(* CoDeSys 2.3.9.16 project: oscat320.pro *)
(* Libraries: Standard.lib 22.11.04 10:21:12 *)

(* PLC configuration (modules and I/O channels)
K-Bus [K_Bus] node 0, in %IB0 out %QB0
Fieldbus variables [FB_VARS] node 1, in %IB0 out %QB0
*)

(* Global variable list: Constants *)
VAR_GLOBAL CONSTANT
	STRING_LENGTH : INT := 250;
	NETWORK_BUFFER_LONG_SIZE : UINT := 3999;
	NETWORK_BUFFER_SHORT_SIZE : UINT := 1459;
END_VAR




(* revisionhistory
hm 3. mar. 2007
	extended accuracy of pi2
	renamed T0 to Tk for better compatibility with other libraries
	renamed C t0 c0 for better compatibility

hm	2. may. 2007
	added RU universal gas constant

hm	1. oct. 2007
	added setup parameter STEP7

hm 31. oct. 2007
	added PN

hm	6. mar. 2008
	added setup Parameter EXTENDED_ASCII

hm	28. Mar. 2008
	added setup parameter STRING_LENGTH

hm	7. apr. 2008
	Deleted unused setup parameter Step7

hm	19. apr. 2008
	added setup parameter NETWORK_BUFFER_SIZE

hm	27. apr. 2008
	added PI05 and PI025

hm	18. may. 2008
	added charname lists
	renamed E to E1

hm	30. jun. 2008
	reduced size of string constants to 253 to avoid problems with target aixia DCUF

hm	21. sep. 2008
	added section language setup
	added section location setup

hm	20. oct. 2008
	changed to structured constants

hm	16. nov. 2008
	moved structured constants to global vars for compatibility reasons

hm	13. nov. 2009
	added network_buffer_short_size
	renamed network_buffer_long_size
	changed string length to 250
*)

(* Global variable list: Globale_Variablen *)
VAR_GLOBAL
	MATH : CONSTANTS_MATH;
	PHYS : CONSTANTS_PHYS;
	LANGUAGE : CONSTANTS_LANGUAGE;
	SETUP : CONSTANTS_SETUP;
	LOCATION : CONSTANTS_LOCATION;
END_VAR

(* Data type *)
TYPE CALENDAR :
STRUCT
	UTC : DT;						(* world time UTC *)
	LDT : DT;						(* local time *)
	LDATE : DATE;				(* local date *)
	LTOD : TOD;					(* local time of day *)
	YEAR : INT;					(* year of LDATE *)
	MONTH : INT;					(* month of LDATE *)
	DAY : INT;						(* day of LDATE *)
	WEEKDAY : INT;				(* weekday of LDATE *)
	OFFSET : INT;					(* Time Zone Offset for Local time in minutes *)
	DST_EN : BOOL;				(* daylight savings time enable *)
	DST_ON : BOOL;				(* true when daylight savings time os on *)
	NAME : STRING(5);			(* name of time zone *)
	LOCATION : INT;				(* location number pls see location setup *)
	LONGITUDE : REAL;			(* longitude of current location *)
	LATITUDE : REAL;			(* latitude of current location *)
	SUN_RISE : TOD;				(* sun_rise for current location *)
	SUN_SET : TOD;				(* sun_set for current location *)
	SUN_MIDDAY : TOD;			(* worldtime when sun stands at south position *)
	SUN_HEIGTH : REAL	;		(* suns heigth at midday, south position *)
	SUN_HOR : REAL;			(* sun angle horizontal 0 = north in degrees *)
	SUN_VER : REAL;			(* sun angle vertical above horizon in degrees *)
	NIGHT : BOOL;				(* true between sun_set and sun_rise *)
	HOLIDAY : BOOL;				(* true when holiday *)
	HOLY_NAME : STRING(30);	(* name of holiday *)
	WORK_WEEK : INT;			(* current work week *)
END_STRUCT
END_TYPE

(* revision history
hm	21. nov. 2008	rev 1.0
	original version

hm	8. feb. 2009	rev 1.1
	added sun position data

hm	10. mar. 2009	rev 1.2
	added work_week, sun_midday, sun_heigth
*)

(* Data type *)
TYPE COMPLEX :
STRUCT
	re : REAL;
	im : REAL;
END_STRUCT
END_TYPE


(* revision history
hm	18. oct. 2008
	original version

*)

(* Data type *)
TYPE CONSTANTS_LANGUAGE :
STRUCT
	(* Language Setup *)
	DEFAULT : INT := 1; (* 1=english, 2=german 3=french *)
	LMAX : INT := 3;
	WEEKDAYS : ARRAY[1..3, 1..7] OF STRING(10) :=	'Monday', 'Tuesday', 'Wednesday', 'Thursday', 'Friday', 'Saturday', 'Sunday',
													'Montag', 'Dienstag', 'Mittwoch', 'Donnerstag', 'Freitag', 'Samstag', 'Sonntag',
													'Lundi', 'Mardi', 'Mercredi', 'Jeudi', 'Vendredi', 'Samedi', 'Dimanche';
	WEEKDAYS2 : ARRAY[1..3, 1..7] OF STRING(2) :=	'Mo', 'Tu', 'We', 'Th', 'Fr', 'Sa', 'Su',
													'Mo', 'Di', 'Mi', 'Do', 'Fr', 'Sa', 'So',
													'Lu', 'Ma', 'Me', 'Je', 'Ve', 'Sa', 'Di';
	MONTHS : ARRAY[1..3, 1..12] OF STRING(10) :=	'January', 'February', 'March', 'April', 'May', 'June', 'July', 'August', 'September', 'October', 'November', 'December',
													'Januar', 'Februar', 'März', 'April', 'Mai', 'Juni', 'Juli', 'August', 'September', 'Oktober', 'November', 'Dezember',
													'Janvier', 'Février', 'mars', 'Avril', 'Mai', 'Juin', 'Juillet', 'Août', 'Septembre', 'Octobre', 'Novembre', 'Decembre';
	MONTHS3 : ARRAY[1..3, 1..12] OF STRING(3) :=	'Jan', 'Feb', 'Mar', 'Apr', 'May', 'Jun', 'Jul', 'Aug', 'Sep', 'Oct', 'Nov', 'Dec',
													'Jan', 'Feb', 'Mrz', 'Apr', 'Mai', 'Jun', 'Jul', 'Aug', 'Sep', 'Okt', 'Nov', 'Dez',
													'Jan', 'Fev', 'Mar', 'Avr', 'Mai', 'Jun', 'Jul', 'Aou', 'Sep', 'Oct', 'Nov', 'Dec';
	DIRS : ARRAY[1..3,0..15] OF STRING(3) :=		'N', 'NNE', 'NE', 'ENE', 'E', 'ESE', 'SE', 'SSE', 'S', 'SSW', 'SW', 'WSW', 'W', 'WNW', 'NW', 'NNW',
													'N', 'NNO', 'NO', 'ONO', 'O', 'OSO', 'SO', 'SSO', 'S', 'SSW', 'SW', 'WSW', 'W', 'WNW', 'NW', 'NNW',
													'N', 'NNO', 'NO', 'ONO', 'O', 'OSO', 'SO', 'SSO', 'S', 'SSW', 'SW', 'WSW', 'W', 'WNW', 'NW', 'NNW';
END_STRUCT
END_TYPE

(* revision history
hm	19. oct. 2008	rev 1.0
	original version

hm	22. oct. 2008	rev 1.1
	added directions DIRS

hm	23. dec. 2008	rev 1.2
	added french language

*)

(* Data type *)
TYPE CONSTANTS_LOCATION :
STRUCT
	(* location setup *)
	DEFAULT : INT := 1; (* 1=germany, 2=austria 3=france *)
	LMAX : INT := 3;

	(*	if month = 0 then F_day is the offset in days from easter
		used :0 = NOT used, 1 = used, -1..-7 menas the weekday before the specified DATE example -3 means wednesday before 23.11
	*)
	HOLIDAY : ARRAY[1..3, 0..29] OF HOLIDAY_DATA := (name := 'Neujahr', day := 1, month := 1, use := 1),
													(name := 'Heilig Drei Könige', day := 6, month := 1, use := 1),
													(name := 'Karfreitag', day := -2, month := 0, use := 1),
													(name := 'Ostersonntag', day := 0, month := 0, use := 1),
													(name := 'Ostermontag', day := 1, month := 0, use := 1),
													(name := 'Tag der Arbeit', day := 1, month := 5, use := 1),
													(name := 'Christi Himmelfahrt', day := 39, month := 0, use := 1),
													(name := 'Pfingstsonntag', day := 49, month := 0, use := 1),
													(name := 'Pfingstmontag', day := 50, month := 0, use := 1),
													(name := 'Fronleichnam', day := 60, month := 0, use := 1),
													(name := 'Augsburger Friedensfest', day := 8, month := 8, use := 0),
													(name := 'Maria Himmelfahrt', day := 15, month := 8, use := 1),
													(name := 'Tag der Deutschen Einheit', day := 3, month := 10, use := 1),
													(name := 'Reformationstag', day := 31, month := 10, use := 0),
													(name := 'Allerheiligen', day := 1, month := 11, use := 1),
													(name := 'Buss und Bettag', day := 23, month := 11, use := 0),
													(name := '1. Weihnachtstag', day := 25, month := 12, use := 1),
													(name := '2. Weihnachtstag', day := 26, month := 12, use := 1),
													(),
													(),
													(),
													(),
													(),
													(),
													(),
													(),
													(),
													(),
													(),
													(),
													(* the next 30 lines are for austrian holidays *)
													(name := 'Neujahr', day := 1, month := 1, use := 1),
													(name := 'Heilig Drei Könige', day := 6, month := 1, use := 1),
													(name := 'Karfreitag', day := -2, month := 0, use := 1),
													(name := 'Ostersonntag', day := 0, month := 0, use := 1),
													(name := 'Ostermontag', day := 1, month := 0, use := 1),
													(name := '', day := 1, month := 5, use := 0),
													(name := 'Christi Himmelfahrt', day := 39, month := 0, use := 1),
													(name := 'Pfingstsonntag', day := 49, month := 0, use := 1),
													(name := 'Pfingstmontag', day := 50, month := 0, use := 1),
													(name := 'Fronleichnam', day := 60, month := 0, use := 1),
													(name := '', day := 8, month := 8, use := 0),
													(name := 'Maria Himmelfahrt', day := 15, month := 8, use := 1),
													(name := '', day := 3, month := 10, use := 0),
													(name := '', day := 31, month := 10, use := 0),
													(name := 'Allerheiligen', day := 1, month := 11, use := 1),
													(name := 'Maria Empfängnis', day := 8, month := 12, use := 1),
													(name := '1. Weihnachtstag', day := 25, month := 12, use := 1),
													(name := '2. Weihnachtstag', day := 26, month := 12, use := 1),
													(),
													(),
													(),
													(),
													(),
													(),
													(),
													(),
													(),
													(),
													(),
													(),
													(* the next 30 lines are for french holidays *)
													(name := 'Nouvel an', day := 1, month := 1, use := 1),
													(name := 'St Valentin', day := 14, month := 2, use := 0),
													(name := 'Vendredi Saint (alsace)', day := -2, month := 0, use := 0),
													(name := 'Dimanche de pâques', day := 0, month := 0, use := 1),
													(name := 'Lundi de pâques', day := 1, month := 0, use := 1),
													(name := 'Jeudi de Ascension', day := 39, month := 0, use := 1),
													(name := 'dimanche de Pentecôte ', day := 49, month := 0, use := 1),
													(name := 'jeudi de la Trinité', day := 60, month := 0, use := 0),
													(name := 'Fête du travail', day := 1, month := 5, use := 1),
													(name := 'Victoire 1945 ', day := 8, month := 5, use := 1),
													(name := 'Prise de La bastille', day := 14, month := 7, use := 1),
													(name := '15 Août 1944', day := 15, month := 8, use := 1),
													(name := 'Halloween', day := 31, month := 10, use := 0),
													(name := 'Armistice 1918', day := 11, month := 11, use := 1),
													(name := 'Noël', day := 25, month := 12, use := 1),
													(name := 'Saint Étienne (alsace)', day := 26, month := 12, use := 0),
													(name := 'Fête de la musique', day := 21, month := 6, use := 0),
													(),
													(),
													(),
													(),
													(),
													(),
													(),
													(),
													(),
													(),
													(),
													(),
													();

END_STRUCT
END_TYPE


(* revision history
hm	20. oct. 2008	rev 1.0
	original version

hm	23. dec. 2008	rev 1.1
	added french holidays
*)

(* Data type *)
TYPE CONSTANTS_MATH :
STRUCT
	PI : REAL := 	3.14159265358979323846264338327950288;	(* Kreiszahl PI *)
	PI2 : REAL := 	6.28318530717958647692528676655900576;	(* PI * 2 *)
	PI4 : REAL :=  12.56637061435917295385057353311801152;	(* PI * 4 *)
	PI05 : REAL :=  1.5707963267949;						(* PI / 2 *)
	PI025 : REAL := 0.785398163397448;						(* PI / 4 *)
	PI_INV : REAL := 0.318309886183791;						(* 1 / PI *)
	E : REAL := 	2.71828182845904523536028747135266249;	(* Eulersche Konstante e *)
	E_INV : REAL := 0.367879441171442;						(* 1 / e *)
	SQ2 : REAL :=	1.4142135623731;						(* Wurzel von 2 *)
END_STRUCT
END_TYPE



(* revision history
hm	26.10.2008	rev 1.0
	original version

*)

(* Data type *)
TYPE CONSTANTS_PHYS :
STRUCT
	C : REAL := 299792458.0;				(* Lichtgeschwindigkeit in m/s *)
	E : REAL := 1.60217653E-19;				(* elementarladung in Colomb = A * s *)
	G : REAL := 9.80665; 						(* Erdbeschleunigung in m / s² *)
	T0 : REAL := -273.15;						(* absoluter Nullpunkt in °C *)
	RU : REAL := 8.314472; 					(* Universelle Gaskonstante in J / (mol · K) *)
	PN : REAL := 101325.0;					(* NormalDruck in Pa *)
END_STRUCT
END_TYPE



(* revision history
hm	18.10.2008	rev 1.0
	original version

hm	13. mar. 2009	rev 1.1
	real constants updated to new systax using dot

*)

(* Data type *)
TYPE CONSTANTS_SETUP :
STRUCT
	(* setup Parameters *)
	EXTENDED_ASCII : BOOL := TRUE;
	CHARNAMES : ARRAY[1..4] OF STRING(253) := ';"&quot;&&amp;<&lt;>&gt;€&euro; &nbsp;¡&iexcl;¢&cent;£&pound;¤&curren;¥&yen;¦&brvbar;§&sect;¨&uml;©&copy;ª&ordf;«&laquo;¬&not;­&shy;®&reg;¯&macr;°&deg;±&plusmn;²&sup2;³&sup3;´&acute;µ&micro;¶&para;·&middot;¸&cedil;¹&sup1;º&ordm;»&raquo;¼&frac14;Û&Ucirc;',
		';¾&frac34;¿&iquest;À&Agrave;Á&Aacute;Â&Acirc;Ã&Atilde;Ä&Auml;Å&Aring;Æ&AElig;Ç&Ccedil;È&Egrave;É&Eacute;Ê&Ecirc;Ë&Euml;Ì&Igrave;Í&Iacute;Î&Icirc;Ï&Iuml;Ð&ETH;Ñ&Ntilde;Ò&Ograve;Ó&Oacute;Ô&Ocirc;Õ&Otilde;Ö&Ouml;×&times;Ø&Oslash;Ù&Ugrave;Ú&Uacute;½&frac12;',
		';Ü&Uuml;Ý&Yacute;Þ&THORN;ß&szlig;à&agrave;á&aacute;â&acirc;ã&atilde;ä&auml;å&aring;æ&aelig;ç&ccedil;è&egrave;é&eacute;ê&ecirc;ë&euml;ì&igrave;í&iacute;î&icirc;ï&iuml;ð&eth;ñ&ntilde;ò&ograve;ó&oacute;ô&ocirc;õ&otilde;ö&ouml;÷&divide;ø&oslash;ù&ugrave;',
		';ú&uacute;û&ucirc;ü&uuml;ý&yacute;þ&thorn;ÿ&yuml;';
	MTH_OFS : ARRAY[1..12] OF INT := 0,31,59,90,120,151,181,212,243,273,304,334;
	DECADES : ARRAY[0..8] OF REAL := 1,10,100,1000,10000,10000,100000,1000000,10000000;
END_STRUCT
END_TYPE

(* revision history
hm	24.10.2008	rev 1.0
	original version

*)

(* Data type *)
TYPE ESR_DATA :
STRUCT
	TYP : BYTE;
	ADRESS : STRING(10);
	DS : DT;
	TS : TIME;
	DATA : ARRAY[0..7] OF BYTE;
END_STRUCT
END_TYPE


(* revision history
hm	18. oct. 2008
	original version

*)

(* Data type *)
TYPE HOLIDAY_DATA :
STRUCT
	NAME : STRING(30);
	DAY : SINT;
	MONTH : SINT;
	USE : SINT;
END_STRUCT
END_TYPE


(* revision history
hm	18. oct. 2008
	original version

*)

(* Data type *)
TYPE NETWORK_BUFFER :
STRUCT
	SIZE : UINT;
	BUFFER : NW_BUF_LONG;
END_STRUCT
END_TYPE


(* revision history
hm	18. oct. 2008
	original version

hm 13. nov. 2009
	use constant network_buffer_long_size

*)

(* Data type *)
TYPE NETWORK_BUFFER_SHORT :
STRUCT
	SIZE : UINT;
	BUFFER : NW_BUF_SHORT;
END_STRUCT
END_TYPE


(* revision history
hm 13. nov. 2009
	original version

*)

(* Data type *)
TYPE
	NW_BUF_LONG  : ARRAY[0..NETWORK_BUFFER_LONG_SIZE] OF BYTE;
END_TYPE

(* Data type *)
TYPE
	NW_BUF_SHORT : ARRAY[0..NETWORK_BUFFER_SHORT_SIZE] OF BYTE;
END_TYPE

(* Data type *)
TYPE REAL2 :
STRUCT
	R1 : REAL;	(* small value *)
	RX : REAL;	(* big value *)
END_STRUCT
END_TYPE


(* revision history
hm	18. oct. 2008
	original version

*)

(* Data type *)
TYPE SDT :
STRUCT
	YEAR : INT;
	MONTH : INT;
	DAY : INT;
	WEEKDAY : INT;
	HOUR : INT;
	MINUTE : INT;
	SECOND : INT;
	MS : INT;
END_STRUCT
END_TYPE


(* revision history
hm	18. oct. 2008
	original version

*)

(* Data type *)
TYPE TIMER_EVENT :
STRUCT
	TYP : BYTE;
	CHANNEL : BYTE;
	DAY : BYTE;
	START : TOD;
	DURATION : TIME;
	LAND : BYTE;
	LOR : BYTE;
	LAST : DWORD;
END_STRUCT
END_TYPE


(* revision history
hm	18. oct. 2008
	original version

*)

(* Data type *)
TYPE URL :
STRUCT
	PROTOCOL : STRING(10);
	USER : STRING(20);
	PASSWORD : STRING(20);
	DOMAIN : STRING(80);
	PORT : WORD;
	PATH : STRING(80);
	QUERY : STRING(40);
	ANCHOR : STRING(40);
END_STRUCT
END_TYPE


(* revision history
hm	18. oct. 2008
	original version

*)

(* Data type *)
TYPE VECTOR_3 :
STRUCT
	X : REAL;
	Y : REAL;
	Z : REAL;
END_STRUCT
END_TYPE


(* revision history
hm	18. oct. 2008
	original version

*)

(* POU PLC_PRG, CFC *)
PROGRAM PLC_PRG
VAR
END_VAR
_CFC_ (* Continuous Function Chart, elements in execution order *)
_END_CFC_
END_PROGRAM

(* POU Logic/generators/SEQUENCE_64, ST *)
FUNCTIONBLOCK SEQUENCE_64
VAR_INPUT
	START : BOOL;
	SMAX : INT;
	PROG : ARRAY[0..63]OF TIME;
	RST : BOOL;
END_VAR
VAR_OUTPUT
	STATE : INT := -1;
	TRIG : BOOL;
END_VAR
VAR
	tx : TIME;
	edge: BOOL;
	last: TIME;
END_VAR


(*
version 1.0	29. jun. 2008
programmer 	hugo
tested by	oscat

sequence generates a sequence of states with a programmable length for each state.

*)
(* read system timer *)
tx := DWORD_TO_TIME(T_PLC_MS());
TRIG := FALSE;

IF RST THEN
	STATE := -1;

(* start sequence *)
ELSIF START AND NOT edge THEN
	STATE := 0;
	last := tx;
	TRIG := TRUE;

(* sequence generator *)
ELSIF (STATE >= 0) THEN
	IF (tx - last) >= PROG[STATE] THEN
		STATE := INC2(STATE, 1, -1, SMAX);
		last := tx;
		TRIG := TRUE;
	END_IF;
END_IF;

edge := START;



(* revision history
hm	29. jun. 2008
	original version

*)
END_FUNCTION_BLOCK

(* POU Engineering/measurements/T_PLC_MS, ST *)
FUNCTION T_PLC_MS : DWORD
VAR CONSTANT
	debug : BOOL := 0;
	N : INT := 0;
	offset : DWORD := 0;
END_VAR
VAR
	tx : TIME;
END_VAR

(*
version 1.2	16. nov 2008
programmer 	hugo
tested by	oscat

T_PLC_MS reads the internal PLC timer and return the time, it has the advantage to be able to set a debug mode 
and speed up the counter to test the plc timer overrun which occurs every 50 days respectively 25 days at siemens S7
this routine also allows to correct the behavior of s7 where the internal plc counter will not count all 32 bits.

*)
tx := TIME();
T_PLC_MS := TIME_TO_DWORD(Tx);
(* hier muss die korrektur für step7 stattfinden
plctime muss den vollen wertebereich von time ausnutzen:
wenn bei step7 time -24tage bis plus 24 tage ist dann muss der timer auch beim überlauf auf -24tage springen 
und auf keinen fall auf 0 !!!!
für siemens muss ein weiterer fb im main eingebunden werden der sicherstellt das alle 32 bits durchgezählt werden.
es kann nur ein fb sein den er muss sich das oberste (32te) bit merken.
oder etwa spring s7 bei überlauf auf -24 tage????? dann wäre keine korrektur nötig.
*)
IF debug THEN
	T_PLC_MS := (SHL(T_PLC_MS,N) OR SHL(DWORD#1,N)-1) + OFFSET;
END_IF;

(* revision history
hm	14.9.2007	rev 1.0
	original version

hm	12. nov 2007	rev 1.1
	added temporaray variable tx because some compilers could not handle time() as an argument

hm	16. nov. 2008	rev 1.2
	initialized constants with 0 for compatibility reasons
*)
END_FUNCTION

(* POU Engineering/signal processing/OFFSET, ST *)
FUNCTION OFFSET : REAL
VAR_INPUT
	X : REAL;
	O1, O2, O3, O4 : BOOL;
	D : BOOL;
END_VAR
VAR_INPUT CONSTANT
	Offset_1 : REAL;
	Offset_2 : REAL;
	Offset_3 : REAL;
	Offset_4 : REAL;
	default : REAL;
END_VAR

(*
version 1.0	12 jan 2007
programmer 	oscat
tested by	oscat

The Function offset adds offsets to an analog signal depending on digital inputs.
all selected offsets are added at the same time.
with the input D a default value instead of the input X can be used.

*) 
IF D THEN OFFSET := default; ELSE OFFSET := X; END_IF;
IF O1 THEN OFFSET := OFFSET + offset_1; END_IF;
IF O2 THEN OFFSET := OFFSET + offset_2; END_IF;
IF O3 THEN OFFSET := OFFSET + offset_3; END_IF;
IF O4 THEN OFFSET := OFFSET + offset_4; END_IF;



(* revision history
hm	12. jan 2007
	original version


*)
END_FUNCTION

(* POU Mathematical/INC2, ST *)
FUNCTION INC2 : INT
VAR_INPUT
	X : INT;
	D : INT;
	L : INT;
	U : INT;
END_VAR
VAR
	tmp: INT;
END_VAR


(*
version 1.0	29. jun. 2008
programmer 	hugo
tested by	oscat

This function increments the input X by the value D and compares the result with U.
if the output exceeds U it will continue to count from L again.

*)
tmp := U - L + 1;
INC2 := (X + D - L + tmp) MOD tmp + L;



(* revision history
hm	29. jun. 2008		REV 1.0
	original version


*)
END_FUNCTION

(* POU Engineering/automation/SRAMP, ST *)
FUNCTIONBLOCK SRAMP
VAR_INPUT
	X : REAL;
	A_UP : REAL;
	A_DN :REAL;
	VU_MAX : REAL;
	VD_MAX : REAL;
	LIMIT_HIGH : REAL;
	LIMIT_LOW : REAL;
	RST : BOOL;
END_VAR
VAR_OUTPUT
	Y : REAL;
	V : REAL;
END_VAR
VAR
	cycle_time : TC_S;
	init: BOOL;
END_VAR


(*
	version 1.1	11. mar. 2009
	programmer 	hugo
	tested by		tobias

RAMPS generates output signal which are slew rate and acceleration controlled.

*)
(* read the system_time in microseconds *)
cycle_time();

(* assure range of inputs *)
A_up := MAX(0.0, A_UP);
A_dn := MIN(0.0, A_dn);
VU_max := MAX(0.0, VU_max);
VD_max := MIN(0.0, VD_MAX);

(* calculate the output offset *)
IF rst OR NOT init THEN
	init := TRUE;
	Y := 0.0;
	V := 0.0;
ELSIF X = Y THEN
	v := 0.0;
ELSIF X > Y THEN
	(* output is too low >> ramp up and brake at the end *)
	(* accelerate the speed and limit to vu_max *)
	v := MIN(v + A_UP * cycle_time.TC, vu_max);
	(* calculate the max speed to be able to brake and select the lowest *)
	v := MIN(SQRT((Y-X) * 2.0 * A_DN), v);
	(* calculate the output and obey limits *)
	y := LIMIT(limit_low, y + MIN(v * cycle_time.TC, X-Y), limit_high);
ELSIF X < Y THEN
	(* output is too high >> ramp dn and brake at the end *)
	(* accelerate the speed and limit to vd_max *)
	v := MAX(v + A_DN * cycle_time.TC, vd_max);
	(* calculate the max speed to be able to brake and select the lowest *)
	v := MAX(-SQRT((Y-X) * 2.0 * A_UP), v);
	(* calculate the output and obey limits *)
	y := LIMIT(limit_low, y + MAX(v * cycle_time.TC, X-Y), limit_high);
END_IF;


(* revision history
hm	13. mar. 2008	rev 1.0
	original version

hm	11. mar. 2009	rev 1.1
	real constants updated to new systax using dot																																																																																																																																																																																																																																																																																																																																																																																																																																																																																																																																																																																																																																																																																																																																																																																																																																																																																																																																																																																																																																																											

*)
END_FUNCTION_BLOCK

(* POU Engineering/measurements/CYCLE_TIME, ST *)
FUNCTION_BLOCK CYCLE_TIME
VAR_INPUT
	RST : BOOL;
END_VAR
VAR_OUTPUT
	ct_min : TIME;
	ct_max : TIME;
	ct_last : TIME;
	systime : TIME;
	sysdays : INT;
	cycles : DWORD;
END_VAR
VAR
	last_cycle : TIME;
	tx: TIME;
	init: BOOL;
END_VAR


(*
	version 1.2	16 sep 2007
	programmer 	hugo
	tested BY		hans

this function block measures the cycle time and displays the last, min and max cycle time of the current task.
the resolution is 1ms.
the cycles output is a dword counter which counts the cycles.
a rst pulse on the input will reset all data.


*)
tx := DWORD_TO_TIME(T_PLC_MS()) - last_cycle;
IF rst THEN
	ct_min := t#10h;
	ct_max := t#0ms;
	cycles := 0;
ELSIF last_cycle > t#0s THEN
	IF tx < ct_min THEN ct_min := tx;
	ELSIF tx > ct_max THEN ct_max := tx;
	END_IF;
	ct_last := tx;
ELSIF ct_min = t#0s THEN
	ct_min := t#0s - t#1ms;
END_IF;
IF init THEN
	systime := systime + tx;
		IF systime >= t#1d THEN
			systime := systime - t#1d;
			sysdays := sysdays + 1;
		END_IF;
END_IF;
init := TRUE;
last_cycle := last_cycle + tx;
cycles := cycles + 1;

(*	revision history
hm 12.12.2006		rev 1.1
	added cycles output, a dword cycle counter.
hm 10.3.2007			rev 1.2
	changed initialization of ct_min to t#10h for compatibility with siemens s7

hm	16.9.2007		rev 1.2
	changed Time() in T_PLC_MS() for compatibility resons

*)
END_FUNCTION_BLOCK

(* POU Engineering/measurements/TC_S, ST *)
FUNCTION_BLOCK TC_S

VAR_OUTPUT
	TC : REAL;
END_VAR
VAR
	init: BOOL;
	tx: DWORD;
	last: DWORD;
END_VAR

(*
	version 1.2	11. mar. 2009
	programmer 	hugo
	tested by		tobias

TC_S delivers the time it was last called on the output TC in seconds.

*)
(* read system timer *)
tx := T_PLC_US();

IF NOT init THEN
	init := TRUE;
	TC := 0.0;
ELSE
	tc := DWORD_TO_REAL(tx - last)*1.0E-6;
END_IF;
last := tx;

(* revision history
hm	13. mar. 2008	rev 1.0
	original version

hm	16. mar 2008	rev 1.1
	added type conversion to avoid warnings under codesys 3.0

hm	11. mar. 2009	rev 1.2
	changed real constants to use dot syntax

*)
END_FUNCTION_BLOCK

(* POU Engineering/measurements/T_PLC_US, ST *)
FUNCTION T_PLC_US : DWORD
VAR CONSTANT
	debug : BOOL := 0;
	N : INT := 0;
	offset : DWORD := 0;
END_VAR
VAR
	tx : TIME;
END_VAR

(*
version 1.2	16 nov 2008
programmer 	hugo
tested by	tobias

T_PLC_US reads the internal PLC timer and return the time, it has the advantage to be able to set a debug mode 
and speed up the counter to test the plc timer overrun which occurs every 50 days respectively 25 days at siemens S7
this routine also allows to correct the behavior of s7 where the internal plc counter will not count all 32 bits.

*)
tx := TIME();
T_PLC_US := TIME_TO_DWORD(Tx)*1000;
(* hier muss die korrektur für step7 stattfinden
plctime muss den vollen wertebereich von time ausnutzen:
wenn bei step7 time -24tage bis plus 24 tage ist dann muss der timer auch beim überlauf auf -24tage springen 
und auf keinen fall auf 0 !!!!
für siemens muss ein weiterer fb im main eingebunden werden der sicherstellt das alle 32 bits durchgezählt werden.
es kann nur ein fb sein den er muss sich das oberste (32te) bit merken.
oder etwa spring s7 bei überlauf auf -24 tage????? dann wäre keine korrektur nötig.
*)
IF debug THEN
	T_PLC_US := (SHL(T_PLC_US,N) OR SHL(DWORD#1,N)-1) + OFFSET;
END_IF;

(* revision history
hm	14.9.2007	rev 1.0
	original version

hm	12. nov 2007	rev 1.1
	added temporaray variable tx because some compilers could not handle time() as an argument

hm	16. nov. 2008	rev 1.2
	initialized constants with 0 for compatibility reasons

*)
END_FUNCTION

(* POU Logic/generators/TMAX, ST *)
FUNCTIONBLOCK TMAX
VAR_INPUT
	IN : BOOL;
	PT : TIME;
END_VAR
VAR_OUTPUT
	Q : BOOL;
	Z : BOOL;
END_VAR
VAR
	tx : TIME;
	start : TIME;
	last_in: BOOL;
END_VAR

(*
version 1.0	20. jul. 2008
programmer 	hugo
tested by	oscat

Q of tmax will follow IN except that it forces a maximum ontime for the output Q.
the output Z will be active for one cycle if the output is forced low by the timeout.

*)
(* read system timer *)
tx := DWORD_TO_TIME(T_PLC_MS());

Z := FALSE;

IF NOT in THEN
	Q := FALSE;
ELSIF IN AND NOT last_in THEN
	Q := TRUE;
	start := tx;
ELSIF (tx - start >= PT) AND Q THEN
	Q := FALSE;
	Z := TRUE;
END_IF;

last_in := IN;



(* revision history
hm	20. jul. 2008	rev 1.0
	original version

*)
END_FUNCTION_BLOCK

(* POU Logic/generators/TMIN, ST *)
FUNCTIONBLOCK TMIN
VAR_INPUT
	IN : BOOL;
	PT : TIME;
END_VAR
VAR_OUTPUT
	Q : BOOL;
END_VAR
VAR
	pm : TP;
END_VAR

(*
version 1.0	21. jul. 2008
programmer 	hugo
tested by	oscat

Q of tMIN will follow IN except that it forces a minimum ontime for the output Q.

*)
pm(in := IN, PT := PT);
Q := IN OR pm.Q;


(* revision history
hm	21. jul. 2008	rev 1.0
	original version

*)
END_FUNCTION_BLOCK

(* POU Logic/generators/TOF_1, ST *)
FUNCTIONBLOCK TOF_1
VAR_INPUT
	IN : BOOL;
	PT : TIME;
	RST : BOOL;
END_VAR
VAR_OUTPUT
	Q : BOOL;
END_VAR
VAR
	tx : TIME;
	start : TIME;
END_VAR

(*
version 1.0	17. jul. 2008
programmer 	hugo
tested by	oscat

TOF_1 will extend a pulse on input in for PT seconds.
in addition the timer can be cleared asynchronously with rst.
TOF_1 is the same function as TOF from the standard LIB except the asynchronous reset input.

*)
(* read system timer *)
tx := DWORD_TO_TIME(T_PLC_MS());

IF RST THEN
	Q := FALSE;
ELSIF IN THEN
	Q := TRUE;
	start := tx;
ELSIF tx - start >= PT THEN
	Q := FALSE;
END_IF;




(* revision history
hm	17. jul. 2008	rev 1.0
	original version

*)
END_FUNCTION_BLOCK

(* POU Logic/generators/TP_1, ST *)
FUNCTIONBLOCK TP_1
VAR_INPUT
	IN : BOOL;
	PT : TIME;
	RST : BOOL;
END_VAR
VAR_OUTPUT
	Q : BOOL;
END_VAR
VAR
	tx : TIME;
	start : TIME;
	ix : BOOL;
END_VAR

(*
version 1.0	28. jun. 2008
programmer 	hugo
tested by		oscat

TP_1 generates a pulse every time it is calles with in := TRUE.
in addition the timer can be cleared asynchronously with rst.
the timer can be retriggered as often as necessary. it will count PT from the last trigger.

*)
(* read system timer *)
tx := DWORD_TO_TIME(T_PLC_MS());

IF RST THEN
	Q := FALSE;
ELSIF IN AND NOT ix THEN
	Q := TRUE;
	start := tx;
ELSIF tx - start >= PT THEN
	Q := FALSE;
END_IF;

ix:= IN;



(* revision history
hm	28. jun. 2008
	original version

*)
END_FUNCTION_BLOCK

(* POU Logic/generators/TP_1D, ST *)
FUNCTIONBLOCK TP_1D
VAR_INPUT
	IN : BOOL;
	PT1 : TIME;
	PTD : TIME;
	RST : BOOL;
END_VAR
VAR_OUTPUT
	Q : BOOL;
	W : BOOL;
END_VAR
VAR
	tx : TIME;
	start: TIME;
	ix: BOOL;
END_VAR


(*
version 1.0	28. jun. 2008
programmer 	hugo
tested by	oscat

TP_1D generates a pulse every time it is calles with in := TRUE.
the module will reset IN by itself so no clearing of in is necessary.
in addition the timer can be cleared asynchronously with rst.
also the rst input is cleared by the module itself.
the timer can be retriggered as often as necessary. it will count PT from the last trigger.
after the time PT1 is elapsed, the timer blocks itself for PT2 and only allow new sequences after PT2 has elapsed.


*)
(* read system timer *)
tx := DWORD_TO_TIME(T_PLC_MS());

IF RST THEN
	Q := FALSE;
	rst := FALSE;
	W := FALSE;
ELSIF W THEN
	IF tx - start >= PTD THEN
		W := FALSE;
	END_IF;
ELSIF IN AND NOT ix THEN
	Q := TRUE;
	start := tx;
	in := FALSE;
ELSIF tx - start >= PT1 THEN
	Q := FALSE;
	W := TRUE;
	start := tx;
END_IF;

ix := IN;



(* revision history
hm	28. jun. 2008
	original version

*)
END_FUNCTION_BLOCK

(* POU Mathematical/Array/_ARRAY_ABS, ST *)
FUNCTION _ARRAY_ABS : BOOL
VAR_INPUT
	pt : POINTER TO ARRAY[0..32000] OF REAL;
	size : UINT;
END_VAR
VAR
	i: UINT;
	stop: UINT;
END_VAR

(*
version 1.0	2. apr. 2008
programmer 	hugo
tested by	tobias

this function will calculate the absolute value of each element of the array and stroe the result instead of the element.
Array[i] := ABS(ARRAY[i]).
the function needs to be called:	array_avg(adr("array"),sizeof("array"));
because this function works with pointers its very time efficient and it needs no extra memory.

*)
stop := SHR(size,2)-1;
FOR i := 0 TO stop DO
	PT^[i] := ABS(PT^[i]);
END_FOR;
_ARRAY_ABS := TRUE;


(* revision history
hm	2. apr 2008		rev 1.0
	original version

*)
END_FUNCTION

(* POU Mathematical/Array/_ARRAY_ADD, ST *)
FUNCTION _ARRAY_ADD : BOOL
VAR_INPUT
	pt : POINTER TO ARRAY[0..32000] OF REAL;
	size : UINT;
	X : REAL;
END_VAR
VAR
	i: UINT;
	stop: UINT;
END_VAR

(*
version 1.0	2. apr. 2008
programmer 	hugo
tested by	tobias

this function will add an offset X to each element of the array and stroe the result instead of the element.
Array[i] := ARRAY[i] + X.
the function needs to be called:	array_avg(adr("array"),sizeof("array"));
because this function works with pointers its very time efficient and it needs no extra memory.

*)
stop := SHR(size,2)-1;
FOR i := 0 TO stop DO
	PT^[i] := PT^[i] + X;
END_FOR;
_ARRAY_ADD := TRUE;


(* revision history
hm	2. apr 2008		rev 1.0
	original version

*)
END_FUNCTION

(* POU Mathematical/Array/_ARRAY_INIT, ST *)
FUNCTION _ARRAY_INIT : BOOL
VAR_INPUT
	pt : POINTER TO ARRAY[0..32000] OF REAL;
	size : UINT;
	init : REAL;
END_VAR
VAR
	i: UINT;
	stop: UINT;
END_VAR


(*
version 1.3	16 mar 2008
programmer 	hugo
tested by		tobias

this function will initialize a given array with a value init.
the function needs to be called:	_array_init(adr("array"),sizeof("array"));
this function will manipulate a given array.
the function manipulates the original array, it rerturnes true when finished.
because this function works with pointers its very time efficient and it needs no extra memory.

*)
stop := SHR(size,2)-1;
FOR i := 0 TO stop DO
	pt^[i] := init;
END_FOR;

_array_init := TRUE;

(* revision History

hm 6.1.2007		rev 1.1
	change type of function to bool
	added  array_init := true to set output true.

hm	14.11.2007	rev 1.2
	changed stop calculation to be more efficient

hm	16.3. 2008		rev 1.3
	changed type of input size to uint
*)
END_FUNCTION

(* POU Mathematical/Array/_ARRAY_MEDIAN, ST *)
FUNCTION _ARRAY_MEDIAN : REAL
VAR_INPUT
	pt : POINTER TO ARRAY[0..32000] OF REAL;
	size : UINT;
END_VAR
VAR
	i: UINT;
	stop: UINT;
END_VAR

(*
version 1.5	16 mar 2008
programmer 	hugo
tested by		tobias

this function will calculate the median of a given array.
in order to do so the ariginal array is sorted and stays sorted after the function finishes
the function needs to be called:	_array_median(adr("array"),sizeof("array"));
this function will manipulate a given array.
the function will return the median of the original array.
for example [12,0,4,7,1] the median is 4 and the array after the function is called is [0,1,4,7,12]
because this function works with pointers its very time efficient and it needs no extra memory.

*)
_ARRAY_SORT(pt,size);
stop := SHR(size,2)-1;
IF EVEN(UINT_TO_INT(stop)) THEN
	_ARRAY_MEDIAN := pt^[SHR(stop,1)];
ELSE
	i := SHR(stop,1);
	_ARRAY_MEDIAN := (pt^[i] + pt^[i+1]) * 0.5;
END_IF;

(* old code
stop := (size - SIZEOF(pt)) / SIZEOF(pt);
FOR i := 0 TO stop - 1 DO
	FOR m := i + 1 TO stop DO
		IF pt^[i] > pt^[m] THEN
			temp := pt^[i];
			pt^[i] := pt^[m];
			pt^[m] := temp;
		END_IF;
	END_FOR;
END_FOR;
IF even(stop) THEN
	_array_median := pt^[stop/2];
ELSE
	i := stop/2;
	_array_median := (pt^[i] + pt^[i+1])/2;
END_IF;
*)
(* revision history
hm 	3.3.2007		rev 1.1
	corrected an error, changed the statement line 14	i := TRUNC(stop/2); to i := stop/2;

hm		22. sep 2007	rev 1.2
	changed algorithm to use _array_soft for performance reasons

hm		8. oct 2007		rev 1.3
	deleted unused variables m and temp

hm		14. nov 2007	rev 1.4
	corrected a problem with size calculation

hm		16.3. 2008		rev 1.5
	changed type of input size to uint
	performance improvements
*)
END_FUNCTION

(* POU Mathematical/Array/_ARRAY_SORT, ST *)
FUNCTION _ARRAY_SORT : BOOL
VAR_INPUT
	pt : POINTER TO ARRAY[1..32000] OF REAL;
	size : UINT;
END_VAR
VAR
	i: INT;
	j: INT;
	temp : REAL;
	stop : INT;
	heapsize: INT;
	popmax : REAL;
	size2: INT;
	hs2: INT;
END_VAR

(*
version 1.6	16. mar. 2008
programmer 	hugo
tested by		tobias

this function will sort a given array.
the function needs to be called:	_array_sort(adr("array"),sizeof("array"));
this function will manipulate a given array.
the function will not return anything except true, it will instead manipulate the original array.
because this function works with pointers its very time efficient and it needs no extra memory.

*)
(* generate heap *)

size := SHR(size,2);
size2 := UINT_TO_INT(SHR(size,1));
FOR i := SIZE2  TO 1 BY -1 DO 		(* zweite Hälfte des Feldes braucht nicht betrachtet werden *)
	j:=i;
    WHILE j <= SIZE2 DO
     	stop := j * 2 + 1;               (* finde Maximum der (beiden) Söhne *)
        IF stop > UINT_TO_INT(SIZE) THEN stop := stop - 1;
        ELSIF pt^[stop-1] > pt^[stop] THEN stop := stop - 1;
		END_IF;
        IF pt^[j] < pt^[stop] THEN   		(* ggf. tauschen *)
         	temp := pt^[j];
            pt^[j] := pt^[stop];
            pt^[stop] := temp;
        END_IF;
        j := stop;
    END_WHILE;
END_FOR;

(* heapsort *)
FOR heapsize := UINT_TO_INT(size) TO 1 BY -1 DO
	popmax := pt^[1];
	pt^[1] := pt^[heapsize];
   	i := 1;
	hs2 := SHR(heapsize,1);
	WHILE i <= hs2 DO	     (* letztes Element an Anfang setzen und versickern lassen *)
       	stop := i * 2 + 1;                (* finde Maximum der (beiden) Söhne *)
        	IF stop > heapsize THEN stop := stop - 1;
        	ELSIF pt^[stop-1] > pt^[stop] THEN stop := stop - 1;
	 	END_IF;
        	IF pt^[i] < pt^[stop] THEN	     (* ggf. tauschen *)
            		temp := pt^[i];
            		pt^[i] := pt^[stop];
            		pt^[stop] := temp;
        	END_IF;
        	i := stop;
    	END_WHILE;
	pt^[heapsize] := popmax;
END_FOR;

_ARRAY_SORT := TRUE;

(* old algorithm bubble sort used before rev 1.2
stop := (size - SIZEOF(pt)) / SIZEOF(pt);
FOR i := 0 TO stop - 1 DO
	FOR m := i + 1 TO stop DO
		IF pt^[i] > pt^[m] THEN
			temp := pt^[i];
			pt^[i] := pt^[m];
			pt^[m] := temp;
		END_IF;
	END_FOR;
END_FOR;
_array_sort := TRUE;

*)
(* revision history

hm 	6.1.2007 	rev 1.1
	changed return value to true

hm	22. sep 2007	rev 1.2
	changed sorting algorithm to heap sort for performance reasons

hm 	14. nov 2007	rev 1.3
	changed calculation of stop to be more efficient

hm	15 dec 2007	rev 1.4
	added function return true

hm	5. jan 2008		rev 1.5
	improved performance

hm	16. mar. 2008	rev 1.6
	changed type of input size to uint

hm	28. mar. 2008	rev 1.7
	changed input f to pt

*)
END_FUNCTION

(* POU Mathematical/EVEN, ST *)
FUNCTION EVEN : BOOL
VAR_INPUT
	in : DINT;
END_VAR


(*
version 1.1	1 dec 2007
programmer 	hugo
tested by		tobias

this function chacks an input for even  value
the output is true if the input is even.
execution time on wago 750 - 841 =  10  us
*)
EVEN := NOT in.0;

(* revision history
hm	1. oct 2006	rev 1.0
	ORIGINAL VERSION

hm	01.12.2007	rev 1.1
	changed code for improved performance

hm	21. mar. 2008	rev 1.2
	changed type of input IN from INT to DINT
*)
END_FUNCTION

(* POU Mathematical/Array/_ARRAY_MUL, ST *)
FUNCTION _ARRAY_MUL : BOOL
VAR_INPUT
	pt : POINTER TO ARRAY[0..32000] OF REAL;
	size : UINT;
	X : REAL;
END_VAR
VAR
	i: UINT;
	stop: UINT;
END_VAR

(*
version 1.0	2. apr. 2008
programmer 	hugo
tested by	tobias

this function will multiply each element of the array and stroe the result instead of the element.
Array[i] := ARRAY[i] * X.
the function needs to be called:	array_avg(adr("array"),sizeof("array"));
because this function works with pointers its very time efficient and it needs no extra memory.

*)
stop := SHR(size,2)-1;
FOR i := 0 TO stop DO
	PT^[i] := PT^[i] * X;
END_FOR;
_ARRAY_MUL := TRUE;


(* revision history
hm	2. apr 2008		rev 1.0
	original version

*)
END_FUNCTION

(* POU Mathematical/Array/_ARRAY_SHUFFLE, ST *)
FUNCTION _ARRAY_SHUFFLE : BOOL
VAR_INPUT
	pt : POINTER TO ARRAY[0..32000] OF REAL;
	size : UINT;
END_VAR
VAR
	temp : REAL;
	pos  : INT;
	i: INT;
	stop: INT;
END_VAR


(*
version 1.2	30. mar. 2008
programmer 	kurt
tested by		hugo

this function will randomly shuffle the elements of an array
*)
stop := UINT_TO_INT(SHR(size,2)-1);
FOR i := 0 TO stop DO
        pos := RDM2(i+pos,0,stop);
        (* swap elements *)
        temp := pt^[i];
        pt^[i] := pt^[pos];
        pt^[pos] := temp;
END_FOR;

_ARRAY_SHUFFLE := TRUE;


(* revision History
hm 	4. mar 2008	rev 1.0
	original version

hm	16. mar. 2008	rev 1.1
	changed type of input size to uint

hm	30. mar. 2008	rev 1.2
	changed last in rdm2 fromm pos to i + pos to allow for more randomness

*)
END_FUNCTION

(* POU Mathematical/RDM2, ST *)
FUNCTION RDM2 : INT
VAR_INPUT
	last : INT;
	low : INT;
	high : INT;
END_VAR


(*
version 1.1	18. oct. 2008
programmer 	hugo
tested by	tobias

this function calculates an integer pseudo random number
the random number will be in the range of low <= rdm2 <= high.

*)
RDM2 := TRUNC(RDM(FRACT(last * math.PI)) * (high - low + 1)) + low;

(* revision history
hm		29. feb 2008		rev 1.0
	original version

hm		18. oct. 2008		rev 1.1
	using math constants

*)
END_FUNCTION

(* POU Mathematical/RDM, ST *)
FUNCTION RDM : REAL
VAR_INPUT
	last : REAL;
END_VAR
VAR
	tn : DWORD;
	tc : INT;
END_VAR


(*
version 1.9	10. mar. 2009
programmer 	hugo
tested by		tobias

this function calculates a pseudo random number
to generate the number it reads the sps timer and calculates a random number between 0 and 1:
in order to use rdm more then once within one sps cycle it need to be called with different seed numbers LAST.

*)
tn := T_PLC_MS();
tc := BIT_COUNT(tn);
tn.31 := tn.2;
tn.30 := tn.5;
tn.29 := tn.4;
tn.28 := tn.1;
tn.27 := tn.0;
tn.26 := tn.7;
tn.25 := tn.6;
tn.24 := tn.3;
tn := ROL(tn,BIT_COUNT(tn)) OR 16#80000001;
tn := tn MOD 71474513 + INT_TO_DWORD(tc + 77);
RDM := FRACT(DWORD_TO_REAL(tn) / 10000000.0 * (math.E - LIMIT(0.0,last,1.0)));


(*
pt := ADR(temp);
pt^ := (T_PLC_MS() AND 16#007FFFFF) OR 16#3D000000;
RDM := fract(modR(temp*e+pi1, PI1-last) + modR(temp*PI1+e + last,e-last));
*)

(* revision history
hm		16. jan 2007		rev 1.0
	original version

hm		11. nov 2007		rev 1.1
	changed time() into t_plc_ms()

hm		20. nov 2007		rev 1.2
	changed code of temp calculation to avoid overflow in modr due to resuclt would not fit DINT for high timeer values

hm		5. jan 2008		rev 1.3
	changed calculation of temp to avoid problem with high values of t_plc_ms

hm		2. feb 2008		rev 1.4
	changed algorithm to avoind non iec functions and guarantee more randomness

hm	10. mar. 2008		rev 1.5
	make sure last will be between 0 and 1 to avoid invalid results

hm	16. mar. 2008		rev 1.6
	added conversion for tc to avoid warnings under codesys 3.0

hm	18. may. 2008		rev 1.7
	changed constant E to E1

hm	18. oct. 2008		rev 1.8
	using math constants

hm	10. mar. 2009		rev 1.9
	real constants updated to new systax using dot

*)
END_FUNCTION

(* POU Logic/gate logic/BIT_COUNT, ST *)
FUNCTION BIT_COUNT : INT
VAR_INPUT
	IN : DWORD;
END_VAR


(*
version 1.1	10 sep 2007
programmer 	hugo
tested by		tobias

BIT_COUNT counts the amount True of bits in a dword.
for exabple: bit_count(3) returns 2 because two bits (bits 0 and 1) are true and all others are false. 

*)
WHILE in > 0 DO
	IF in.0 THEN Bit_Count := Bit_Count + 1; END_IF;
	in := SHR(in,1);
END_WHILE;



(* revision history
5.7.2007	rev 1.0		original version

10.9.2007	rev 1.1		hm
	changed algorithm for better performace
	the execution time has reduced by a factor of 5
	deleted unused variable temp
*)
END_FUNCTION

(* POU Mathematical/FRACT, ST *)
FUNCTION FRACT : REAL
VAR_INPUT
	x : REAL;
END_VAR


(*
version 1.3	10. mar. 2009
programmer 	hugo
tested by		tobias

this function returns the fraction of a real number
fract(3.14) = 0.14

*)
IF ABS(x) < 2.0E9 THEN
	FRACT := x - DINT_TO_REAL(D_TRUNC(x));
ELSE
	FRACT := 0.0;
END_IF;

(* revision history
hm	4. aug 2006	rev 1.0
	original version

hm	11. mar 2008	rev 1.1
	added dint_to_real for compatibility reasons
	now returns 0 for number > 2e9
	changed input to x

hm	21. mar. 2008	rev 1.2
	use D_trunc instead of TRUNC for compatibility reasons

hm	10. mar. 2009	rev 1.3
	real constants updated to new systax using dot

*)
END_FUNCTION

(* POU Mathematical/D_TRUNC, ST *)
FUNCTION D_TRUNC : DINT
VAR_INPUT
	X : REAL;
END_VAR

(*
version 1.2	10. mar. 2009
programmer 	hugo
tested by		oscat

d_trunc truncates a real to a dint 1.5 will be 1 and -1.5 will be -1
d_trunc is necessary because many systems do not offer a trunc to a dint
also real_to_dint will not deliver the same result on different systems

*)
D_TRUNC := REAL_TO_DINT(X);
IF X > 0.0 THEN
	IF DINT_TO_REAL(D_TRUNC) > X THEN D_TRUNC := D_TRUNC - 1; END_IF;
ELSE
	IF DINT_TO_REAL(D_TRUNC) < X THEN D_TRUNC := D_TRUNC + 1; END_IF;
END_IF;


(* for systems that support a dint truncation this routine can be replaced by trunc() *)


(* revision history
hm	21. mar. 2008	rev 1.0
	original version

hm	31. oct. 2008	rev 1.1
	optimized performance

hm	10. mar. 2009	rev 1.2
	real constants updated to new systax using dot
*)
END_FUNCTION

(* POU Buffer Management/_BUFFER_CLEAR, ST *)
FUNCTION _BUFFER_CLEAR : BOOL
VAR_INPUT
	PT : POINTER TO BYTE;
	SIZE : UINT;
END_VAR
VAR
	ptw : POINTER TO DWORD;
	temp: DWORD;
	end, end32 : DWORD;
END_VAR


(*
version 1.2	31. oct. 2008
programmer 	hugo
tested by	oscat

this function will initialize a given array of byte with 0.
the function needs to be called:	_buffer_clear(adr("array"),sizeof("array"));
this function will manipulate a given array.
the function manipulates the original array, it rerturnes true when finished.
because this function works with pointers its very time efficient and it needs no extra memory.

*)
(* this routine uses 32 bit access to gain speed *)
(* first access bytes till pointer is aligned for 32 bit access *)
temp := pt;
end := temp + UINT_TO_DWORD(size);
end32 := end - 3;
WHILE (pt < end) AND ((temp AND 16#00000003) > 0) DO
	pt^ := 0;
	pt := pt + 1;
	temp := temp + 1;
END_WHILE;
(* pointer is aligned, now copy 32 bits at a time *)
ptw := pt;
WHILE ptw < end32 DO (* *)
	ptw^ := 0;
	ptw := ptw + 4;
END_WHILE;
(* copy the remaining bytes in byte mode *)
pt := ptw;
WHILE pt < end DO
	pt^ := 0;
	pt := pt + 1;
END_WHILE;

_BUFFER_CLEAR := TRUE;

(* revision History
hm 	5. mar. 2008	rev 1.0
	original version

hm	16. mar. 2008	rev 1.1
	added type conversion to avoid warnings under codesys 30
	chaged type of input size to uint
	deleted unused variable i

hm	31. oct. 2008	rev 1.2
	corrected an error while routine would write outside of arrays

*)
END_FUNCTION

(* POU Buffer Management/_BUFFER_INIT, ST *)
FUNCTION _BUFFER_INIT : BOOL
VAR_INPUT
	PT : POINTER TO BYTE;
	SIZE : UINT;
	INIT : BYTE;
END_VAR
VAR
	ptw : POINTER TO DWORD;
	temp : DWORD;
	end, end32 : DWORD;
END_VAR


(*
version 1.2	31. oct. 2008
programmer 	hugo
tested by	oscat

this function will initialize a given array of byte with init.
the function needs to be called:	_buffer_init(adr("array"),sizeof("array"),init);
this function will manipulate a given array.
the function manipulates the original array, it rerturnes true when finished.
because this function works with pointers its very time efficient and it needs no extra memory.

*)
(* this routine uses 32 bit access to gain speed *)
(* first access bytes till pointer is aligned for 32 bit access *)
temp := pt;
end := temp + UINT_TO_DWORD(size);
end32 := end - 3;
WHILE (pt < end) AND ((temp AND 16#00000003) > 0) DO
	pt^ := init;
	pt := pt + 1;
	temp := temp + 1;
END_WHILE;
(* pointer is aligned, now copy 32 bits at a time *)
ptw := pt;
temp := SHL(BYTE_TO_DWORD(init),24) OR SHL(BYTE_TO_DWORD(init),16) OR SHL(BYTE_TO_DWORD(init),8) OR BYTE_TO_DWORD(init);
WHILE ptw < end32 DO
	ptw^ := temp;
	ptw := ptw + 4;
END_WHILE;
(* copy the remaining bytes in byte mode *)
pt := ptw;
WHILE pt < end DO
	pt^ := init;
	pt := pt + 1;
END_WHILE;

_BUFFER_INIT := TRUE;

(* revision History
hm 	5. mar. 2008	rev 1.0
	original version

hm	16. mar. 2008	rev 1.1
	added type conversion to avoid warnings under codesys 3.0
	chaged type of input size to uint.

hm	31. oct. 2008	rev 1.2
	corrected an error while routine would write outside of arrays

*)
END_FUNCTION

(* POU Buffer Management/_BUFFER_INSERT, ST *)
FUNCTION _BUFFER_INSERT : BOOL
VAR_INPUT
	STR : STRING(STRING_LENGTH);
	POS : INT;
	PT : POINTER TO ARRAY[0..32767] OF BYTE;
	SIZE : UINT;
END_VAR
VAR
	end : INT;
	lx: INT;
	i: INT;
END_VAR


(*
version 1.4	12. nov. 2009
programmer 	hugo
tested by		oscat

this function will initialize a given array of byte with init.
the function needs to be called:	_buffer_init(adr("array"),sizeof("array"),init);
this function will manipulate a given array.
the function manipulates the original array, it rerturnes true when finished.
because this function works with pointers its very time efficient and it needs no extra memory.

*)
lx := LEN(str);
end := pos + lx;
(* first move the upper part of the buffer to make space for the string *)
FOR i := UINT_TO_INT(size) - 1 TO end BY -1 DO
	pt^[i] := pt^[i-lx];
END_FOR;
(* copy the string *)
_BUFFER_INSERT := _STRING_TO_BUFFER(str, pos, PT, size);


(* revision History
hm 	9. mar. 2008	rev 1.0
	original version

hm	16. mar. 2008	rev 1.1
	changed type of input size to uint

hm	13. may. 2008	rev 1.2
	changed type of pointer to array[1..32767]
	changed size of string to STRING_LENGTH

hm	23. mar. 2009	rev 1.3
	avoid writing to input pos

hm	12. nov. 2009	rev 1.4
	code optimized

*)
END_FUNCTION

(* POU Buffer Management/_STRING_TO_BUFFER, ST *)
FUNCTION _STRING_TO_BUFFER : BOOL
VAR_INPUT
	STR : STRING(STRING_LENGTH);
	POS : INT;
	PT : POINTER TO ARRAY[0..32767] OF BYTE;
	SIZE : UINT;
END_VAR
VAR
	ps : POINTER TO BYTE;
	i: INT;
	end: INT;
END_VAR


(*
version 1.3	12. nov. 2009
programmer 	hugo
tested by		oscat

this function will copy a string into an array of byte starting at position pos.
the function needs to be called:	_String_To_buffer(str, pos, adr("array"),sizeof("array"));
this function will manipulate the array directly in memory and returns true when finished.
because this function works with pointers its very time efficient and it needs no extra memory.

*)
ps := ADR(str);
end := MIN(pos + LEN(str), UINT_TO_INT(size));
IF end > 0 THEN end := end -1; END_IF;
FOR i := pos TO end DO
	pt^[i] := ps^;
	ps := ps + 1;
END_FOR;

_STRING_TO_BUFFER := TRUE;

(* revision History

hm 	5. mar. 2008	rev 1.0
	original version

hm	16. mar. 2008	rev 1.1
	changed type of input size to uint

hm	13. may. 2008	rev 1.2
	changed type of pointer to array[1..32767]
	changed size of string to STRING_LENGTH

hm	12. nov. 2009	rev 1.3
	limit end to size - 1

*)
END_FUNCTION

(* POU Engineering/signal generators/_RMP_B, ST *)
FUNCTION_BLOCK _RMP_B
VAR_INPUT
	DIR : BOOL;  (* true = up *)
	E : BOOL := TRUE;
	TR : TIME;
END_VAR
VAR_IN_OUT
	RMP : BYTE;
END_VAR
VAR
	tx, tl : DWORD;
	step : INT;
	init: BOOL;
	last_dir: BOOL;
END_VAR


(*
version 1.1	20. nov. 2008
programmer 	hugo
tested by	oscat


_RMP_B generates a ramp on an external var of type byte
tr is the total ramp time, E is an enable and dir the direction of the ramp

*)
tx := T_PLC_MS();
IF E AND init THEN
	(* we need to set tl = tx when direction changes *)
	IF dir XOR last_dir THEN
	 tl := tx;
	 last_dir := dir;
	END_IF;
	(* check_elapsed time and calculate only if necessary *)
	IF tr > t#0s THEN
		step := DWORD_TO_INT(SHL(tx-tl, 8) / TIME_TO_DWORD(TR));
	ELSE
		step := 255;
	END_IF;
	IF step > 0 THEN
		(* perform the step on the ramp *)
		tl := tx;
		(* calculate the step response *)
		IF NOT dir THEN step := - step; END_IF;
		rmp := INT_TO_BYTE(LIMIT(0, BYTE_TO_INT(rmp) + step, 255));
	END_IF;
ELSE
	tl := tx;
	init := TRUE;
END_IF;


(* revison history
hm	22. oct. 2008	rev 1.0
	original version

hm	20. nov. 2008	rev 1.1
	set default for E to be TRUE
	added init

*)
END_FUNCTION_BLOCK

(* POU Engineering/signal generators/_RMP_NEXT, ST *)
FUNCTION_BLOCK _RMP_NEXT
VAR_INPUT
	E : BOOL := TRUE;
	IN : BYTE;
	TR : TIME;
	TF : TIME;
	TL : TIME;
END_VAR
VAR_OUTPUT
	DIR : BOOL;    (* upwards = TRUE *)
	UP : BOOL;
	DN : BOOL;
END_VAR
VAR_IN_OUT
	OUT : BYTE;
END_VAR
VAR
	rmx : _RMP_B;
	dirx : TREND_DW;
	t_lock :TP;
	xen: BOOL;
	xdir: BOOL;
END_VAR


(*
version 1.4	18. jul. 2009
programmer 	hugo
tested by		oscat


_RMP_NEXT  will generate a ramp output following the input IN.
on a rising ramp the output will stop as soon as it has surpassed the input in, and on a falling ramp it will stop when out is smaller than in.
a lockout time T_L will be added between up and down direction.

*)
dirx(X := in);

t_lock(in := FALSE, pt := TL);

IF dirx.TU AND (OUT < IN) THEN
	IF NOT xdir AND xen THEN t_lock(in := TRUE); END_IF;
	xen := TRUE;
	xdir := TRUE;
ELSIF dirx.TD AND (OUT > IN) THEN
	IF xdir AND xen THEN t_lock(in := TRUE); END_IF;
	xen := TRUE;
	xdir := FALSE;
ELSIF xen THEN
	IF (xdir AND (out >= in)) OR (NOT xdir AND (out <= in)) THEN
		xen := FALSE;
		IF tl > t#0s THEN t_lock(IN := TRUE); END_IF;
	END_IF;
END_IF;

IF NOT t_lock.Q AND xen THEN
		UP := XDIR;
		DIR := XDIR;
		DN := NOT XDIR;
ELSE
	UP := FALSE;
	DN := FALSE;
END_IF;

rmx(rmp := OUT, E := E AND (UP OR DN) , dir := DIR, tr := SEL(dir, TF, TR));


(* revison history
hm	23. nov. 2008	rev 1.0
	original version

hm	24. jan. 2009	rev 1.1
	deleted unused vars tmp1, tmp2

hm	20. feb. 2009	rev 1.2
	improved algorithm
	added TL

hm	9. mar. 2009	rev 1.3
	input E was ignored
	removed double assignments

hm	18. jul. 2009	rev 1.4
	improved performance

*)
END_FUNCTION_BLOCK

(* POU Engineering/signal processing/TREND_DW, ST *)
FUNCTION_BLOCK TREND_DW
VAR_INPUT
	X : DWORD;
END_VAR
VAR_OUTPUT
	Q : BOOL;
	TU : BOOL;
	TD : BOOL;
	D : DWORD;
END_VAR
VAR
	last_X: DWORD;
END_VAR

(*
version 1.2	14. mar. 2009
programmer 	hugo
tested by		oscat

trend_DW analyses the trend of a input signal.
The Output Q is True if the input X is >= last_X and is false if the input X is <= last_X
in addition to the trend the output TU will be high for one cycle to signal a rising of the input value X
and  TD will signal a decreasing value on the input X.
in case of a change the output D will show the delta of the input to the last input value.


*)
IF X > last_X THEN
	TU := TRUE;
	TD := FALSE;
	D := X - last_X;
	Q := TRUE;
ELSIF X < last_X THEN
	TD := TRUE;
	TU := FALSE;
	D := last_X - X;
	Q := FALSE;
ELSE
	TU := FALSE;
	TD := FALSE;
	D := 0;
END_IF;
last_X := X;



(* revision history
hm	21. nov. 2008	rev 1.0
	original version

hm	20. feb. 2009	rev 1.1
	added outputs TU, TD and D

hm	14. mar. 2009	rev 1.2
	removed double assignments

*)
END_FUNCTION_BLOCK

(* POU Engineering/signal generators/_RMP_W, ST *)
FUNCTION_BLOCK _RMP_W
VAR_INPUT
	DIR : BOOL;
	E : BOOL := TRUE;
	TR : TIME;
END_VAR
VAR_IN_OUT
	RMP : WORD;
END_VAR
VAR
	tx, tl : DWORD;
	step : DINT;
	init: BOOL;
	last_dir : BOOL;
END_VAR


(*
version 1.1	20. nov. 2008
programmer 	hugo
tested by	oscat


_RMP_B generates a ramp on an external var of type byte
tr is the total ramp time, E is an enable and dir the direction of the ramp

*)
tx := T_PLC_MS();
IF E AND init THEN
	(* we need to set tl = tx when direction changes *)
	IF dir XOR last_dir THEN
	 tl := tx;
	 last_dir := dir;
	END_IF;
	(* check_elapsed time and calculate only if necessary *)
	IF tr > t#0s THEN
		step := DWORD_TO_DINT(SHL(tx-tl, 16) / TIME_TO_DWORD(TR));
	ELSE
		step := 65535;
	END_IF;
	IF step > 0 THEN
		(* perform the step on the ramp *)
		tl := tx;
		(* calculate the step response *)
		IF NOT dir THEN step := - step; END_IF;
		rmp := DINT_TO_WORD(LIMIT(0, WORD_TO_DINT(rmp) + step, 65535));
	END_IF;
ELSE
	tl := tx;
	init := TRUE;
END_IF;


(* revison history
hm	22. oct. 2008	rev 1.0
	original version

hm	20. nov. 2008	rev 1.1
	set default for E to be TRUE
	added init

*)
END_FUNCTION_BLOCK

(* POU Logic/generators/A_TRIG, ST *)
FUNCTION_BLOCK A_TRIG
VAR_INPUT
	IN : REAL;
	RES : REAL;
END_VAR
VAR_OUTPUT
	Q : BOOL;
	D : REAL;
END_VAR
VAR
	last_in : REAL;
END_VAR

(*
version 1.1	25. oct. 2008
programmer 	hugo
tested by	oscat

this block is similar to the IEC Standard R_trig and F_trig but it monitors a REAL for change.
if the valiue on IN changes more then D from the last value it will generate trigger and display the difference in output D.
the trigger will only be active for one cycle.

*)
D := IN - LAST_IN;
Q := ABS(D) > res;
IF Q THEN last_in := IN; END_IF;
D := IN - LAST_IN;


(* revision history

hm 	16. jul. 2008	rev 1.0
	original version released

hm	25. oct. 2008	rev 1.1
	code optimization
	a_trig now also works for res = 0

*)
END_FUNCTION_BLOCK

(* POU Mathematical/ACOSH, ST *)
FUNCTION ACOSH : REAL
VAR_INPUT
	X : REAL;
END_VAR


(*
version 1.3	10. mar. 2009
programmer 	hugo
tested by		tobias

this function calculates the arcus cos hyperbolicus

*)
ACOSH := LN(SQRT(X * X - 1.0) + X);

(* revision history
hm		12 jan 2007	rev 1.0
	original version

hm		2. dec 2007	rev 1.1
	changed code for better performance

hm	16. mar. 2007		rev 1.2
	changed sequence of calculations to improve performance

hm	10. mar. 2009		rev 1.3
	real constants updated to new systax using dot

*)
END_FUNCTION

(* POU Mathematical/ACOTH, ST *)
FUNCTION ACOTH : REAL
VAR_INPUT
	X : REAL;
END_VAR


(*
version 1.2	10. mar. 2009
programmer 	hugo
tested by		tobias

this function calculates the arcus cotangens hyperbolicus

*)
ACOTH := LN((x+1.0)/(x-1.0))*0.5;

(* revision history
hm		12 jan 2007	rev 1.0
	original version

hm		5. jan 2008	rev 1.1
	improved code for better performance

hm	10. mar. 2009		rev 1.2
	real constants updated to new systax using dot

*)
END_FUNCTION

(* POU Building/actuators/ACTUATOR_2P, ST *)
FUNCTION_BLOCK ACTUATOR_2P
VAR_INPUT
	IN : BYTE;
	TEST : BOOL;
	ARE : BOOL := TRUE;
END_VAR
VAR_IN_OUT
	ARX : BOOL;
END_VAR
VAR_INPUT CONSTANT
	CYCLE_TIME : TIME;
	SENS : BYTE;
	SELF_ACT_TIME : TIME;
	SELF_ACT_PULSE : TIME;
	SELF_ACT_CYCLES : INT := 1;
END_VAR
VAR_OUTPUT
	OUT : BOOL;
	ARO : BOOL;
END_VAR
VAR
	timer : AUTORUN;
	pwgen : GEN_PULSE;
END_VAR


(*
version 2.1	24. jan. 2009
programmer 	hugo
tested by		oscat

this is an intelligent actuator interface for any 2point actuator like coil drive.
the 2Point actuator can only switch on/off and therefore the input must be converted to on/off cycles.
the interface can be programmed with double click on the symbol.
in addition a self_act_time and self_act_cycles ca be programmed to switch n times on/off every self_act_time to avoid a valve to freeze.
the input value must be between 0 and 255. with the setup variable sens one can specify what must be the minimum input to turn the valve on at all.
at the same time an input > 255-sens will turn the valve on at all times.


*)
(* run the autorun timer *)
timer(trun := SELF_ACT_PULSE * (2 * SELF_ACT_CYCLES), toff := SELF_ACT_TIME, Test := TEST, ARE := ARE, arx := ARX);
ARO := timer.ARO;

(* run the pulse width generator *)
IF aro THEN
	pwgen(PTL := SELF_ACT_PULSE, PTH := SELF_ACT_PULSE);
	out := pwgen.Q;
ELSIF in < sens THEN
	out := FALSE;
ELSIF in > BYTE#255 - sens THEN
	out := TRUE;
ELSE
	pwgen.PTH := (CYCLE_TIME * BAND_B(IN,SENS)) / 255;
	pwgen.PTL := CYCLE_TIME - pwgen.PTH;
	pwgen();
	out := pwgen.Q;
END_IF;



(* revision history
hm	7.10.2006 		rev 1.1
	changed error pos could not reach 1 or 0 under certain conditions due to error in code.
	changed on and off in force and force_in for better usability.

hm	17.1.2007		rev 1.2
	deleted unused variable time_overflow

hm	15.9.2007		rev 1.3
	replaced time() with T_PLC_MS for compatibility and performance reasons

hm	19. 11 2007		rev 1.4
	replaced left over statement time() with tx

hm	27. 12. 2007	REV 1.5
	CHANGED CODE FOR BETTER PERFORMANCE

hm	21. oct. 2008	rev 1.6
	code optimized

hm	23. nov. 2008	rev 2.0
	new code using library modules

hm	24. jan. 2009	rev 2.1
	deleted unused var inb
*)
END_FUNCTION_BLOCK

(* POU Building/actuators/AUTORUN, ST *)
FUNCTION_BLOCK AUTORUN
VAR_INPUT
	IN : BOOL;
	TEST : BOOL;
	ARE : BOOL := TRUE;
END_VAR
VAR_IN_OUT
	ARX : BOOL;
END_VAR
VAR_INPUT CONSTANT
	TRUN : TIME;
	TOFF : TIME;
END_VAR
VAR_OUTPUT
	OUT : BOOL;
	ARO : BOOL;
END_VAR
VAR
	timer : _RMP_B;
	val : BYTE;
END_VAR



(*
version 1.0	20. nov 2008
programmer 	hugo
tested by	oscat




*)
(* run the integrator when T_off > T#0s *)
IF TOFF > T#0s THEN
	timer(DIR:= OUT, TR := SEL(OUT, TOFF, TRUN), RMP := val);
ELSE
	val := 255;
END_IF;


(* when timer = 0 or test then initiate autorun until timer reaches 255 *)
IF (NOT ARX AND ARE AND val = 0) OR TEST THEN
	val := 0;
	ARO := TRUE;
	ARX := TRUE;
ELSIF val = 255 AND ARO THEN
	ARO := FALSE;
	ARX := FALSE;
END_IF;

(* output is true when autorun ARO is true or in = TRUE *)
out := IN OR ARO;



(* revision history
hm 20. nov. 2008	rev 1.0
	original version

*)
END_FUNCTION_BLOCK

(* POU Engineering/signal generators/GEN_PULSE, ST *)
FUNCTION_BLOCK GEN_PULSE
VAR_INPUT
	ENQ : BOOL := TRUE;
	PTH : TIME;
	PTL : TIME;
END_VAR
VAR_OUTPUT
	Q : BOOL;
END_VAR
VAR
	tx: TIME;
	tn: TIME;
	init: BOOL;
END_VAR

(*
version 1.3	13. nov. 2009
programmer 	hugo
tested by		oscat

GEN_PULSE uses the internal sps timer to generate a continuous output waveform with programmable high and low time.
the accuracy of gen_pulse is depending on the system timer.
when time is 0 the high and low times are exactly one cycle.
ENQ = TRUE will start and ENQ = FALSE will stop the generator.

*)
(* read system timer *)
IF enq THEN
	tx := DWORD_TO_TIME(T_PLC_MS());
	IF NOT init THEN init := TRUE; tn := tx; END_IF;
	IF tx >= tn THEN
		Q := NOT Q;
		tn := tn + SEL(Q,PTL,PTH);
	END_IF;
ELSE
	Q := FALSE;
	init := FALSE;
END_IF;



(* revision history
hm	29. jun. 2008	rev 1.0
	original version

hm	23. nov. 2008	rev 1.1
	set default for enq to be true

hm	18. jul. 2009	rev 1.2
	improved performance

hm	13. nov. 2009	rev 1.3
	corrected error

*)
END_FUNCTION_BLOCK

(* POU Engineering/control/BAND_B, ST *)
FUNCTION BAND_B : BYTE
VAR_INPUT
	X : BYTE;
	B : BYTE;
END_VAR



(*
version 1.0	21. Nov. 2008
programmer 	hugo
tested by	oscat

BAND_B will limit X to B <= X <= 255-B. while X < B the resulkt will be 0 and while X > 255-B the output will be 255
otherwise the result = X.

*)
IF X < B THEN
	BAND_B := 0;
ELSIF X > BYTE#255-B THEN
	BAND_B := 255;
ELSE
	BAND_B := X;
END_IF;



(* revision history
hm	21. nov. 2008	rev 1.0
	original version

*)
END_FUNCTION

(* POU Building/actuators/ACTUATOR_3P, ST *)
FUNCTION_BLOCK ACTUATOR_3P
VAR_INPUT
	in : REAL;
	force : BOOL;
	on : BOOL;
	end_pos : BOOL;
	diag : BOOL;
END_VAR
VAR_INPUT CONSTANT
	min_ontime : TIME := t#10s;
	min_offtime : TIME := t#10s;
	max_runtime : TIME := t#60s;
	auto_diag_time : TIME := t#10d;
	cal_runtime : TIME := t#600s;
	switch_available: BOOL;
END_VAR
VAR_OUTPUT
	out1 : BOOL;
	out2 : BOOL;
	pos : REAL;
	busy : BOOL;
	error : BOOL;
END_VAR
VAR
	val: REAL;
	tx : TIME;
	last_diag: TIME;
	last : TIME;
	runtime_1 : TIME;
	runtime_2 : TIME;
	state : INT;
	rout: FT_RMP;
	end : R_TRIG;
	cal_timer: TIME;
	Tn: TIME;
END_VAR


(*
version 1.3	 15 sep 2007
programmer 	hugo
tested by	oscat

actuator_3P is an interface for a 3 point actuator.
a 3P actuator is a motor with 2 directions that drives a valve or flap. the position of the valve or flap is controlled by runtime of the motor foreward or backward.
the available inputs are:
in is a real value which specifies the position of the actuator, 0 = 0% and 1 = 100% any value <0 or > 1 is limited to 0 or 1.
a force input must be low for normal operation and if switched high, the motor can only be controlled for 0% or 100% positions with the on input.
an and pos input is available for a end_pos switch, this switch indicates the valve or flap to be at either 0% or 100%
a diag input can at any time start a diag cycle which turns the motor towards the 0% position, then measures the runtime to 100% and then the runtime to 0%
these runtimes are stored and used for absolute positioning of the motor during normal operation.
a setup constand "auto_diag_time can be used to specify how often the actuator repeates this auto_diag cycla automatically.
at power on a cycle is perfomed automatically.
a 0 for this value means auto diag is never performed.

the outputs ar out1 and out2 for up and down direction of the motor. to avoid flickering the output can be programmed for min_ontime and min_offtime.
a pos outout indicates the absulute position of the actuator during operation and a busy output indicates the actuator is busy.
a error output is initiated when the specified max_runtime is reached by any direction during debug.
also when the up and down direction differs by more then 10% the error output is set.

for absolute positioning accuracy the actuator has a setup variable "cal_runtime" if this is set the actuator measures the total runtime of the motors and when this 
cal_runtime is exceeded it resets the actuator to 0% position and sets the output again to assure absolute accuracy.

autodiag and calibration can be shut off by setting the appropriate values to 0.
a switch_available setup variable specifies if end_pos switches are available.

*)
(* setup *)
Tn := DWORD_TO_TIME(T_PLC_MS());
tx := Tn - last;
end(clk := end_pos);

(* init only when first started *)
IF state = 0 THEN
	runtime_1 := max_runtime;
	runtime_2 := max_runtime;
	state := 1;
	rout(KR := 1000 / TIME_TO_REAL(runtime_1), KF := 1000 / TIME_TO_REAL(runtime_1) );
	tx := t#0s;
	last := Tn;
	last_diag := last;
END_IF;

(* check for end_sw and stop if reached *)
IF switch_available AND out1 AND end.Q THEN
	(* upper limit has been reached *)
	out1 := 0;
	rout(rmp := 0, in := 1);
	rout.Rmp := 1;
ELSIF switch_available AND out2 AND end.Q THEN
	(* lower limit has been reached *)
	out2 := 0;
	rout(rmp := 0, in := 0);
	rout.Rmp := 1;
END_IF;

(* check for min_offtime and min_ontime and return if it has not elapsed *)
IF NOT busy AND tx < min_offtime THEN
	RETURN;
ELSIF busy AND tx < min_ontime THEN
	RETURN;

(* check for last diag cycle and start diag if auto_diag_time has elapsed *)
ELSIF (tn - last_diag > auto_diag_time AND state > 10 AND auto_diag_time > t#0s) OR (diag AND state >= 10) THEN state := 1;

(* check if force pin is high *)
ELSIF force THEN state := 10;

(* check if calibration is necessary *)
ELSIF cal_timer > cal_runtime AND state = 99 AND cal_runtime > t#0s THEN state := 20;
END_IF;

(* state machine for operation *)
CASE state OF

1 :	(* diagnostic start *)
	(* all data is reset and out2 is turned on to make sure we start from top position *)
	last_diag := tn;
	diag := 0;
	state := 2;
	pos := 0;
	busy := 1;
	last := tn;
	out1 := 0;
	out2 := 1;
	RETURN;

2:	(* wait for max_runtime or end_pos to be reached *)
	IF tx < max_runtime AND NOT end.Q THEN RETURN; END_IF;
	state := 3;
	last := tn;
	out1 := 1;
	out2 := 0;
	RETURN;

3: 	(* measure runtime_2 *)
	IF tx < max_runtime AND NOT end.Q THEN RETURN; END_IF;
	state := 4;
	runtime_1 := tx;
	last := tn;
	out1 := 0;
	out2 := 1;
	RETURN;

4:	(* measure runtime_1 *)
	IF tx < max_runtime AND NOT end.Q THEN RETURN; END_IF;
	state := 99;
	runtime_2 := tx;
	last := tn;
	out2 := 0;
	busy := 0;
	(* reset the output ramp generator to the 0% position as the valve is after diags *)
	rout(rmp := 0, in := 0);
	rout.Rmp := 1;
	cal_timer := t#0s;
	IF DIFFER(TIME_TO_REAL(runtime_1), TIME_TO_REAL(runtime_2), TIME_TO_REAL(max_runtime) * 0.1) THEN error := TRUE;
	ELSIF runtime_1 > MULTIME(max_runtime, 0.9) AND switch_available THEN error := TRUE;
	ELSIF runtime_2 > MULTIME(max_runtime, 0.9) AND switch_available THEN error := TRUE;
	END_IF;
	RETURN;

10: (* force pin is active, outputs are forced on or off by the on pin *)
	IF on AND NOT out2 THEN val := 1;
	ELSIF NOT on AND NOT out1 THEN val := 0;
	END_IF;
	IF NOT force THEN state := 99; END_IF;

20 : (* calibrate to allow for correction of positioning error addig up *)
	cal_timer := t#0s;
	state := 21;
	pos := 0;
	busy := 1;
	last := tn;
	out1 := 0;
	out2 := 1;
	RETURN;

21:	(* after end_sw or max_runtime we can be sure to have reached the 0% position *)
	IF tx < max_runtime AND NOT end.Q THEN RETURN; END_IF;
	state := 99;
	out2 := 0;
	busy := 0;
	last := tn;
	rout(rmp := 0, in := 0);
	rout.Rmp := 1;
	RETURN;

99: (* normal operation *)
	(* only if input changes for an equivalent of min_ontime then change the output *)
	(* if there is a directional change then wait until last step is finished *)
	IF in < TIME_TO_REAL(min_ontime)/TIME_TO_REAL(max_runtime)/2 THEN val := 0;
	ELSIF in > 1 - TIME_TO_REAL(min_ontime)/TIME_TO_REAL(max_runtime)/2 THEN val := 1;
	ELSIF differ(LIMIT(0,in,1), val, TIME_TO_REAL(min_ontime) / TIME_TO_REAL(max_runtime)) OR in = 0 OR in = 1 THEN
		IF in < val AND NOT out1 THEN val := in;
		ELSIF in > val AND NOT out2 THEN val := in;
		END_IF;
	END_IF;

END_CASE;

(* output ramp generator *)
rout(in := val);
out1 := rout.busy AND rout.UD;
out2 := rout.busy AND NOT rout.UD;
pos := rout.out;

(* set the busy output and if busy goes low, then set the last time in order to check for min_offtime *)
IF NOT busy AND rout.busy THEN
	last := tn;
ELSIF busy AND NOT rout.busy THEN
	cal_timer := cal_timer + tx;
	last := tn;
END_IF;
busy := rout.busy;



(* revision history

19.10.2006	rev 1.1
	added security checks for end_switch to avoid overrun of the end_switch, hans

23.1.2007		rev 1.2
	deleted unused variables force_on and force_off

15.9.2007	hm	rev 1.3
	replaced Time() with T_PLC_MS for compatibility and performance reasons

*)
END_FUNCTION_BLOCK

(* POU Mathematical/functions/FT_RMP, ST *)
FUNCTION_BLOCK FT_RMP
VAR_INPUT
	Rmp : BOOL := TRUE;
	in : REAL;
	KR : REAL;
	KF : REAL;
END_VAR
VAR_OUTPUT
	out : REAL;
	busy : BOOL;
	UD : BOOL;
END_VAR
VAR
	tx: TIME;
	last: TIME;
	init: BOOL;
END_VAR

(*
	version 1.4	25 jan 2008
	programmer 	oscat
	tested BY		oscat

this ramp function follows an input signal with a linear ramp up or down, the up or down speed can be set with KF and KR.
a K factor of 1 means 1 unit per second on the output. K factors can only be positive and not negative.
a busy output signals the ramp is running or busy false means the in value is present on the output.
a rmp input false means the output follows the input dierctly while a rmp = true means the output follows the input with a ramp.
a updn output signal the directon of the ramp (up or down).

*)
(* read system time *)
tx := DWORD_TO_TIME(T_PLC_MS()) - last;

IF NOT init THEN
	init := TRUE;
	last := tx;
	tx := t#0s;
	out := in;
END_IF;
IF NOT rmp THEN
	out := in;
	busy := FALSE;
ELSIF out > in THEN
	(* ramp down *)
	out := out - TIME_TO_REAL(tx) * 0.001 * KF;
	out := MAX(in, out);
ELSIF out < in THEN
	(* ramp up *)
	out := out + TIME_TO_REAL(tx) * 0.001 * KR;
	out := MIN(in, out);
END_IF;

(* set busy and dir flags *)
IF out < in THEN
	busy := TRUE;
	ud := TRUE;
ELSIF out > in THEN
	busy := TRUE;
	ud := FALSE;
ELSE
	busy := FALSE;
END_IF;
last := last + tx;


(* revision history:

hm 8.10.2006			rev 1.1
	added ud output

hm 12. feb 2007		rev 1.2
	added init variable and corrected a possible startup problem

hm	17. sep 2007	rev 1.3
	replaced time() with t_plc_ms() for compatibility reasons

hm	25. jan 2008	rev 1.4
	performance improvements
	allow KR and KF to be 0
*)
END_FUNCTION_BLOCK

(* POU Mathematical/DIFFER, ST *)
FUNCTION DIFFER : BOOL
VAR_INPUT
	in1 : REAL;
	in2 : REAL;
	X : REAL;
END_VAR


(*
version 1.1	16 mar 2008
programmer 	hugo
tested by		tobias

this function checks if in1 differs more then x from in2
the output is true if abs(in1-in2) > X

*)
DIFFER := ABS(in1 - in2) > X;

(* revision history
hm		8. oct 2006		rev 1.0
	original version

hm		16. mar 2008	rev 1.1
	improverd code for performance

*)
END_FUNCTION

(* POU Time&Date/MULTIME, ST *)
FUNCTION MULTIME : TIME
VAR_INPUT
	t : TIME;
	M : REAL;
END_VAR


(*
version 1.1	14 mar 2008
programmer 	hugo
tested by		tobias

multiplies a time by a real number and returns a time
*)
MULTIME := DWORD_TO_TIME(REAL_TO_DWORD(DWORD_TO_REAL(TIME_TO_DWORD(t))*M));

(* revision history
hm		2. oct 2006	rev 1.0
	original version

hm		14. mar 2008	rev 1.1
	rounded the result after the last digit

*)
END_FUNCTION

(* POU Building/actuators/ACTUATOR_A, ST *)
FUNCTION_BLOCK ACTUATOR_A
VAR_INPUT
	I1 : BYTE;
	IS : BOOL;
	I2 : BYTE;
	RV : BOOL;
	DX : BOOL;
END_VAR
VAR_INPUT CONSTANT
	RUNTIME : TIME;
	SELF_ACT_TIME : TIME;
	OUT_MIN : WORD;
	OUT_MAX : WORD;
END_VAR
VAR_OUTPUT
	Y : WORD;
END_VAR
VAR
	timer : CYCLE_4;
	dx_edge: BOOL;
END_VAR


(*
version 1.0 8. nov. 2008	
programmer 	hugo
tested by	oscat

ACTUATOR_A drives any valve or similar with 0 - 255 continuous control input.
 
*)
(* run the system timer, if self_act_time = t#0s then state is set to 0 *)
timer(T0 := RUNTIME, T1 := RUNTIME, T3 := SELF_ACT_TIME, sl := DX AND NOT dx_edge, sx := 0, S0 := SELF_ACT_TIME > t#0s);
dx_edge := dx;

CASE timer.STATE OF
	0: 	(* self act min value *)
		Y := OUT_MIN;
	1:	(* self_act max value *)
		Y := OUT_MAX;
	3:	(* normal operation *)
		IF rv THEN
			Y := OUT_MAX - (OUT_MAX - OUT_MIN) * SEL(IS, I1, I2) / 255;
		ELSE
			Y := (OUT_MAX - OUT_MIN) * SEL(IS, I1, I2) / 255 + OUT_MIN;
		END_IF;
END_CASE;




(*
hm 	8. nov. 2008	rev 1.0
	original version

*)
END_FUNCTION_BLOCK

(* POU Logic/generators/CYCLE_4, ST *)
FUNCTION_BLOCK CYCLE_4
VAR_INPUT
	E : BOOL := TRUE;
	T0, T1, T2, T3 : TIME;
	S0 : BOOL;
	SX : INT;
	SL : BOOL;
END_VAR
VAR_OUTPUT
	STATE : INT;
END_VAR
VAR
	tx : TIME;
	last : TIME;
	init: BOOL;
END_VAR


(*
version 1.0	
programmer 	hugo
tested by	oscat


 
*)
(* read system timer *)
tx := DWORD_TO_TIME(T_PLC_MS());
(* init on first cycle *)
IF NOT init THEN
	init := TRUE;
	last := tx;
END_IF;

IF E THEN
	IF SL THEN
		(* when sx > 0 then the state sx is forced to start *)
		state:= LIMIT(0,SX,3);
		last := tx;
		(* this is to avoid to reset sx from the calling programm it does work fine on codesys but i am not sure about other systems, because we are writing to an input *)
		SL := FALSE;
	ELSE
		CASE state OF
			0 :	(* wait for T0 and switch to next cycle *)
				IF tx - last >= T0 THEN
					state := 1;
					last := tx;
				END_IF;
			1 : (* wait for T1 over 1st cycle *)
				IF tx - last >= T1 THEN
					state := 2;
					last := tx;
				END_IF;
			2 : (* wait for T1 over 1st cycle *)
				IF tx - last >= T2 THEN
					state := 3;
					last := tx;
				END_IF;
			3 : (* wait for T2 over 2nd cycle *)
				IF tx - last >= T3 THEN
					IF S0 THEN State := 0; END_IF; (* if S0 is false, the sequence stops at state 3 *)
					last := tx;
				END_IF;
		END_CASE;
	END_IF;
ELSE
	state := 0;
	last := tx;
END_IF;



(*
hm	3. nov. 2008	rev 1.0
	original version

*)
END_FUNCTION_BLOCK

(* POU Building/actuators/ACTUATOR_COIL, ST *)
FUNCTION_BLOCK ACTUATOR_COIL
VAR_INPUT
	IN : BOOL;
END_VAR
VAR_INPUT CONSTANT
	self_act_cycle : TIME := t#10d;
	self_act_time : TIME := t#1s;
END_VAR
VAR_OUTPUT
	OUT :BOOL;
	STATUS : BYTE;
END_VAR
VAR
	last : DWORD;
	init: BOOL;
	tx: DWORD;
	now: DWORD;
END_VAR


(*
version 1.0	1. jun. 2008
programmer 	hugo
tested by		tobias

this is an intelligent actuator interface for any coil actuator.
the coil actuator can only switch on/off.
coil actuators like vents can get stuck if they are not u8sed for a long time and need to be autoactivated on ce in a while.

*)
(* read system time *)
now := T_PLC_MS();

(* initialize for first cycle *)
IF NOT init THEN
	last := now;
	init := TRUE;
ELSIF IN THEN
	OUT := TRUE;
	STATUS := 101; (* activated by input *)
	LAST := now;
ELSE
	OUT := FALSE;
	STATUS := 100; (* disabled *)
	(* now we need to check for self activation *)
	tx := now - last;
	IF (self_act_cycle > T#0s) AND (tx >= TIME_TO_DWORD(self_act_cycle)) THEN
		OUT := TRUE;
		STATUS := 102; (* auto activation *)
		IF tx >= TIME_TO_DWORD(self_act_cycle + self_act_time) THEN
			last := now;
			OUT := FALSE;
			STATUS := 100; (* idle *)
		END_IF;
	END_IF;
END_IF;



(*
revision history:

hm		1. jun. 2008 	rev 1.0
	original version

*)
END_FUNCTION_BLOCK

(* POU Building/actuators/ACTUATOR_PUMP, ST *)
FUNCTION_BLOCK ACTUATOR_PUMP
VAR_INPUT
	IN : BOOL;
	MANUAL : BOOL;
	RST : BOOL;
END_VAR
VAR_INPUT CONSTANT
	MIN_ONTIME : TIME := t#10s;
	MIN_OFFTIME : TIME := t#10s;
	RUN_EVERY : TIME := t#10000m;
END_VAR
VAR_OUTPUT
	PUMP : BOOL;
END_VAR
VAR_IN_OUT
	RUNTIME : UDINT;
	CYCLES : UDINT;
END_VAR
VAR
	tx : TIME;
	last_change : TIME;
	meter : ontime;
	old_man : BOOL;
	init: BOOL;
END_VAR

(*
version 1.4		21. oct. 2008
programmer 		oscat
tested BY		oscat

actuator_pump is a pump interface which can be controlled by an input in and an input manual.
in or manual high turns the pump output on.
a rst input is used to reset the runtime counters.
when the pump was not active for a time run_every the actuator turns on the pump automatically for min_ontime.
two setup variables min_ontime and min_offtime guarantee a minimum runtime and offtime of the pump.
the units are hours and the output type is real to prevent from overfow.

*)
tx := DWORD_TO_TIME(T_PLC_MS());

IF NOT init THEN
	init := TRUE;
	last_change := tx;
ELSIF rst THEN
	rst := FALSE;
	runtime := 0;
	cycles := 0;
ELSIF manual AND NOT pump AND NOT old_man THEN
	last_change := tx;
	pump := TRUE;
ELSIF NOT manual AND old_man AND pump AND NOT in THEN
	last_change := tx;
	pump := FALSE;
ELSIF in AND NOT pump AND tx - last_change >= min_offtime THEN
	last_change := tx;
	pump := TRUE;
ELSIF pump AND NOT in AND NOT manual AND tx - last_change >= min_ontime THEN
	last_change := tx;
	pump := FALSE;
ELSIF NOT pump AND (tx - last_change >= run_every) AND (run_every > T#0s) THEN
	last_change := tx;
	pump := TRUE;
END_IF;

meter(in := pump, seconds := runtime, cycles := cycles);
old_man := manual;



(*
hm	27.12.2006		rev 1.1
	fixed a failure while the pump would run for tmin after startup.

hm	15.9.2007		rev 1.2
	replaced Time() with T_PLC_MS for compatibility and performance reasons

hm	13. oct. 2008	rev 1.3
	auto activation can now be disabled when run_every = t#0s

hm	21. oct. 2008	rev 1.4
	changed to use ontime rev 2.0

*)
END_FUNCTION_BLOCK

(* POU Engineering/automation/MANUAL, ST *)
FUNCTION MANUAL : BOOL
VAR_INPUT
	IN : BOOL;
	ON : BOOL;
	OFF : BOOL;
END_VAR


(*
version 1.0	21. nov. 2008
programmer 	hugo
tested by	oscat

MANUAL is a manual override for digital signals.
when on and off = FALSE, the output follows IN.
ON = TRUE forces the output high, and OFF = TRUE forces the output low.


*)
MANUAL := NOT OFF AND (IN OR ON);



(* revision history
hm	21. nov 2008	rev 1.0
	original version


*)
END_FUNCTION

(* POU Engineering/measurements/METER, ST *)
FUNCTION_BLOCK METER
VAR_INPUT
	M1, M2 : REAL;
	I1, I2 : BOOL;
	D : REAL := 1.0;
	RST : BOOL;
END_VAR
VAR_IN_OUT
	MX : REAL;
END_VAR
VAR
	MR : REAL2;
	MX1, MX2 : REAL; (* current consumption value on M1 and M2 *)
	tx: DWORD;
	last: DWORD;
	tc: REAL;
	init: BOOL;
END_VAR

(*
	version 1.4	8. mar. 2009
	programmer 	oscat
	tested BY	oscat

METER measures usage of power or similar values the output MX is the sum of the inputs over time.
MX := sum over time of (I1 * P1 + I2 * P2)/D.
a simple example is the consumption counter for a 2 stage oil burner where stage 1 is 10KW and stage 2 is 20KW.
I1 and I2 decide which value is accounted for, I1 = True only counts P1, I2 is True counts P2 
and I1 and I2 is true counts P1 and P2.
the meter can be used for all kind of consumption meters. P1 and P2 can change on the fly.

*)
(* measure the last cycle time and make sure we onle execute once every millisecond *)
tx := T_PLC_MS();
IF NOT init THEN
	init := TRUE;
	last := tx;
	mr.RX := mx;
	mr.R1 := 0.0;
ELSIF tx = last THEN
	RETURN;
ELSE
	tc := DWORD_TO_REAL(tx - last) * 0.001;
END_IF;
last := tx;

(* reset *)
IF rst THEN
	mr.R1 := 0.0;
	mr.RX := 0.0;
ELSE
	(* current consumption measurement *)
	IF I1 THEN MX1 := M1; ELSE MX1 := 0.0; END_IF;
	IF I2 THEN MX2 := M2; ELSE MX2 := 0.0; END_IF;
	(* add up the current values in a double real *)
	MR := R2_ADD(MR,(SEL(I1,0.0,mx1) + SEL(I2, 0.0, mx2)) / D * TC);
	(* set the current output value *)
	MX := mr.RX;
END_IF;




(* revision history

hm	16. sep.2007		rev 1.0
	original version

hm	7. feb 2008		rev 1.1
	use new version of ft_int to avoid a counting stop at high values
	deleted unnecessary limits

hm	24. mar. 2008	rev 1.2
	use data_type real2 to extend accuracy to 15 digits total
	do not use ft_int which adds unnecessary overhead

hm	8. feb. 2009	rev 1.3
	changed mx to be I/O
	make sure calculation works for cycle times < 1 ms

hm	8. mar. 2009	rev 1.4
	last was not updated
	code improvements

*)
END_FUNCTION_BLOCK

(* POU Mathematical/Double Precision/R2_ADD, ST *)
FUNCTION R2_ADD : REAL2
VAR_INPUT
	X : Real2;
	Y : REAL;
END_VAR
VAR
	temp: REAL;
END_VAR

(*
version 1.0	20. mar. 2008
programmer 	hugo
tested by	tobias

R2_add adds a real to a double real which extends the accuracy of a real to twice as many digits

*)
temp := X.RX;
R2_ADD.RX := Y + X.R1 + X.RX;
R2_ADD.R1 := temp - R2_ADD.RX + Y + X.R1;


(* revision history
hm		20.3.2008	rev 1.0
	original version

*)
END_FUNCTION

(* POU Engineering/measurements/ONTIME, ST *)
FUNCTION_BLOCK ONTIME
VAR_INPUT
	IN : BOOL;
	RST : BOOL;
END_VAR
VAR_IN_OUT
	SECONDS : UDINT;
	CYCLES : UDINT;
END_VAR
VAR
	tx: DWORD;
	last : DWORD;
	edge : BOOL;
	init: BOOL;
	ms: DWORD;
END_VAR

(*
version 2.3	17. dec. 2008
programmer 	oscat
tested by	tobias

ONTIME measures the ontime of a signal in seconds.
the output SECONDS is of type DWORD which results in a total measurement range of 1 second up to 136 years.
internally ontime works with a resolution of milliseconds

*)
(* read system time *)
tx := T_PLC_MS();

(* make sure the first cycle works correctly *)
IF NOT init OR rst THEN
	init := TRUE;
	last := tx;
	SECONDS := 0;
	CYCLES := BOOL_TO_UINT(in);
	ms := 0;
ELSIF IN THEN
	(* add the current milliseconds *)
	ms := (tx - last) + ms;
	IF ms >= 1000 THEN
		seconds := seconds + 1;
		ms := ms - 1000;
	END_IF;
	cycles := cycles + BOOL_TO_UINT(NOT edge);
END_IF;
last := tx;
edge := in;


(* revision history
hm 22.2.2007		rev 1.1
	changed VAR RETAIN PERSISTENT to VAR RETAIN for better compatibility
	wago lon contollers do not support persisitent

hm 2.8.2007		rev 1.2
	adding time up in a real number will automatically lead to the point where 
	small time scales like the cycle time will be below the resolution of real and therefore
	ontime would not increase in small steps as necessary
	the time is now measured internally in two  dwords and be converted to real only for
	output purposes.
	deleted the variable power because it was unnecessary

hm	16.9.2007		rev 1.3
	changes time() to T_plc_ms() for compatibility reasons

hm	2. dec. 2007	rev 1.4
	chaged code for better performance

hm	16. mar. 2008	rev 1.5
	added type conversions to avoid warnings under codesys 3.0

hm	21. oct. 2008	rev 2.0
	changed module for much better performance and allow for external result storage

hm	10. nov. 2008	rev 2.1
	increased internal resolution to milliseconds

hm	16. nov. 2008	rev 2.2
	changed typecast to avoid warnings

hm	17. dec. 2008	rev 2.3
	fixed an error when in would be true for more then 49 days
*)
END_FUNCTION_BLOCK

(* POU Building/actuators/ACTUATOR_UD, ST *)
FUNCTION_BLOCK ACTUATOR_UD
VAR_INPUT
	UD : BOOL;
	ON : BOOL;
	Manual : BOOL;
	Up : BOOL;
	Dn : BOOL;
	off : BOOL;
	YUP_in : BOOL;
	YDN_in : BOOL;
END_VAR
VAR_INPUT CONSTANT
	TON : TIME;
	TOFF : TIME;
	out_return : BOOL;
END_VAR
VAR_OUTPUT
	Yup : BOOL;
	Ydn : BOOL;
	status : BYTE;
END_VAR
VAR
	tx : TIME;
	last : TIME;
	init: BOOL;
END_VAR

(*
version 1.3	17. oct. 2008
programmer 	hugo
tested by		tobias

out_ud is a up/dn or Right/left locked output driver.
it can be controlled by automatic inputs UD and ON as well as manual inputs for up and dn.
a security input to shut off at any time is prvided by the off input.
two time set inputs ton and toff specify a minimum on time for outputs and a minimum off time before the next output can become active.
the module assures that only one output can be active at any time.
for higher security pls make sure you use hardware locking of the outputs to prevent from defective wiring or outputs.
further security is provided b feedback inputs Yup_in and Ydn_in which are separate inputs for the output signal, if these inputs are not available 
pls connect them directly to Yup and Ydn.
manual mode will override automatic mode by setting the manual input high.
a status output will be 0 for normal operation or 1 - 99 for error reporting and 101 - 199 for status reporting
The status output is ESR comptible.
*)
(* read system time *)
tx := DWORD_TO_TIME(T_PLC_MS());

IF NOT init THEN
	(* INITIALIZATION AT FIRST CALL *)
	last := tx;
	init := TRUE;
ELSIF off THEN
	(* emergency shut off detected *)
	Yup := FALSE;
	ydn := FALSE;
	last := tx;
	status := 101;

(* Watch FOR MIN TON TIME *)
ELSIF ((Yup OR Ydn) AND tx - last < Ton) THEN
	RETURN;
ELSIF NOT yup AND NOT ydn AND tx - last < toff THEN
	RETURN;

(* manual operation *)
ELSIF manual THEN
	status := 102;
	(* directional chage set both outs 0 first *)
	IF yup AND NOT up OR ydn AND NOT dn THEN
		ydn := FALSE;
		yup := FALSE;
		last := tx;
	(* manual up operation *)
	ELSIF UP AND NOT DN AND NOT OFF THEN
		Ydn := FALSE;
		Yup := TRUE;
		last := tx;
		status := 103;
	(* manual down operation *)
	ELSIF DN AND NOT UP AND NOT OFF THEN
		Yup := FALSE;
		Ydn := TRUE;
		last := tx;
		status := 104;
	(* maual mode but no up or down *)
	ELSE
		IF YUP OR YDN THEN LAST := tx; END_IF;
		Yup := FALSE;
		ydn := FALSE;
	END_IF;

(* automatic operation *)
ELSE
	(* directional change set outputs low first *)
	IF yup AND NOT ud OR ydn AND UD THEN
		yup := FALSE;
		ydn := FALSE;
		last := tx;
	(* automatic up operation *)
	ELSIF Ud AND on AND NOT OFF THEN
		Ydn := FALSE;
		Yup := TRUE;
		last := tx;
		status := 111;

	(* automatic down operation *)
	ELSIF NOT UD AND on AND NOT OFF THEN
		Yup := FALSE;
		Ydn := TRUE;
		last := tx;
		status := 112;
	(* standby mode *)
	ELSE
		IF Yup OR Ydn THEN last := tx; END_IF;
		Yup := FALSE;
		Ydn := FALSE;
		status := 110;
	END_IF;
END_IF;

(* make sure Yup and Ydn are never on at the same time *)
IF Ydn AND Yup_in AND out_return THEN
	Ydn := FALSE;
	status := 1;
END_IF;
IF Yup AND Ydn_in AND out_return THEN
	Yup := FALSE;
	status := 2;
END_IF;



(* revision history
hm 22. jan 2007	rev 1.1
	added status output
	changed inputs ton, toff to config variables
	added config var out_return to enable yup_in and Ydn_in
	manual mod will override automatic mode 

hm	15.9.2007	rev 1.2
	replaced Time() with T_PLC_MS for compatibility and performance reasons

hm	17. oct. 2008	rev 1.3
	deleted unnecessary initialization with 0
*)
END_FUNCTION_BLOCK

(* POU Mathematical/AGDF, ST *)
FUNCTION AGDF : REAL
VAR_INPUT
	X : REAL;
END_VAR


(*
version 1.1	10. mar. 2009
programmer 	hugo
tested by		tobias

this function calculates the inverse Gudermannian function.

*)
AGDF := LN((1.0 + SIN(X)) / COS(X));

(* comment
the current implementation gives sufficient accuracy only up to X = 1.57 or an output > 10.
is X closer to PI/2 then the function is more and more unreliable
*)



(* revision history
hm	27. apr. 2008	rev 1.0
	original version

hm	10. mar. 2009	rev 1.1
	real constants updated to new systax using dot

*)
END_FUNCTION

(* POU Engineering/signal processing/AIN, ST *)
FUNCTION AIN : REAL
VAR_INPUT
	in : DWORD;
END_VAR
VAR_INPUT CONSTANT
	Bits : BYTE;
	sign : BYTE := 255;
	low : REAL;
	high : REAL := 10.0;
END_VAR
VAR CONSTANT
	ff : DWORD := 16#FFFFFFFF;
END_VAR
VAR
	temp1 : DWORD;
	temp2 : DWORD;
	sx : BOOL;
END_VAR

(*
version 1.5	16 mar 2008
programmer 	oscat
tested by		tobias

Ain converts signals from A/D converters or other digital sources to an internal real value
the lowest number of bits are extracted from the input word and the sign will be extracted if available separately.
the output signal is then conditioned to range from low to high values for a 0 to max value on the analog inputs:
for example a 15bit input (bits := 12) with sign at bit 15 (0..15) will deliver 0.0 (low value at 0) for an input value of 2#0000_0000_0000
an input value of 2#1111_1111_1111 will deliver 10.0 on the output (high value set to 10).

*) 
(* extract the sign bit *)
IF sign < 32 THEN
	temp1 := SHR(in,sign);
	sx := temp1.0;
ELSE
	sx := FALSE;
END_IF;
temp1 := SHR(ff, 32-bits);
temp2 := in AND temp1;
AIN := (high - low) * DWORD_TO_REAL(temp2) / DWORD_TO_REAL(temp1) + low;
IF sx THEN AIN := -AIN; END_IF;

(* revision history
hm 18.8.2006	rev 1.1
	fixed an error with low value negative and high value 0.

hm 19.1.2007	rev 1.2
	fixed an error with sign bit.

hm	13.9.2007	rev 1.3
	changed code to avoid warning under codesys 2.8.1

hm	2. dec 2007	rev 1.4
	changed code for better performance

hm	16. mar 2008	rev 1.5
	added type conversions to avoid warnings under codesys 30
*)
END_FUNCTION

(* POU Engineering/signal processing/AIN1, ST *)
FUNCTION_BLOCK AIN1
VAR_INPUT
	in : DWORD;
END_VAR
VAR_INPUT CONSTANT
	sign_bit : INT := 255;
	error_bit : INT := 255;
	error_code_en : BOOL;
	error_code : DWORD;
	overflow_bit : INT := 255;
	overflow_code_en : BOOL;
	overflow_code : DWORD;
	Bit_0 : INT;
	Bit_N : INT := 31;
	out_min : REAL;
	out_max : REAL := 10.0;
	code_min : DWORD;
	code_max : DWORD := 16#FFFFFFFF;
	error_output : REAL;
	overflow_output : REAL := 10.0;
END_VAR
VAR_OUTPUT
	out : REAL;
	sign : BOOL;
	error : BOOL;
	overflow : BOOL;
END_VAR
VAR
	tB: DWORD;
END_VAR

(*
version 1.3	10. mar. 2009
programmer 	oscat
tested by		tobias

Ain1 converts signals from A/D converters or other digital sources to an internal real value.

*) 
(* extract error bit *)
error := ((SHR(in,error_bit) AND 16#0000_0001) = 1) OR (error_code_en AND error_code = in);
IF error THEN
	out := error_output;
	RETURN;
END_IF;

(* strip off the data input *)
tb := SHR(SHL(in, 31 - bit_N), 31 - bit_N + Bit_0);

(* extract overflow bit *)
overflow := ((SHR(in,overflow_bit) AND 16#0000_0001) = 1) OR (overflow_code_en AND overflow_code = in) OR (tb < code_min OR tb > code_max);
IF overflow THEN
	out := overflow_output;
	RETURN;
END_IF;

(* extract sign bit *)
sign := (SHR(in,sign_bit) AND 16#0000_0001) = 1;

(* convert in to out *)
out := (DWORD_TO_REAL(tb - code_min) * (out_max - out_min) / DWORD_TO_REAL(code_max - code_min) + out_min);
IF sign THEN out := out * -1.0; END_IF;



(* revision history
hm	23. feb 2008	rev 1.0
	original version

hm	16. mar 2008	rev 1.1
	added type conversions to avoid warnngs under codesys 30

hm	22. apr. 2008	rev 1.2
	corrected error in formula when code_min was set
	corrected error when sign bit was used
	optimized code for better performance

hm	10. mar. 2009	rev 1.3
	real constants updated to new systax using dot

*)
END_FUNCTION_BLOCK

(* POU Building/HLK/AIR_DENSITY, ST *)
FUNCTION AIR_DENSITY : REAL
VAR_INPUT
	T : REAL;
	P : REAL;
	RH : REAL;
END_VAR
VAR CONSTANT
	RL : REAL := 287.05;
	RX : REAL := 3.773319E-3;
END_VAR


(*
version 1.3	13. mar. 2009
programmer 	hugo
tested by		tobias

this function calculates the air density between 0 and 100 deg C

*)
AIR_DENSITY := phys.PN * (1.0 - RH * SDD(T, TRUE) * RX / P) / (RL * ( T - phys.T0));

(* original code used for rev 1.0

SDD := SDD(T,FALSE);
RF := RL / (1- RH*SDD/P*RX);
Air_density := P / (RF * (T-TK));

*)

(* revision history

hm	29.10.2007	rev 1.0
	original version

hm	4.12.2007		rev 1.1
	changed code for better performance

hm	18. oct. 2008	rev 1.2
	using phys constants

hm	13. mar. 2009	rev 1.3
	real constants updated to new systax using dot

*)
END_FUNCTION

(* POU Building/HLK/SDD, ST *)
FUNCTION SDD : REAL
VAR_INPUT
	T : REAL;
	ICE: BOOL;
END_VAR


(*
version 1.1	2 dec 2007
programmer 	hugo
tested by		tobias

this function calculates the vapor saturation pressure for moist Air over ice or water

*)
IF ice THEN
	SDD := 611.153 * EXP(22.4433 * T / (272.186 + T));
ELSE
	SDD := 611.213 * EXP(17.5043 * T / (241.2 + T));
END_IF;



(* revision history

hm 29 oct 2007		rev 1.0
	original version

hm	2. dec 2007		rev 1.1
	changed code for better performance
*)
END_FUNCTION

(* POU Building/HLK/AIR_ENTHALPY, ST *)
FUNCTION AIR_ENTHALPY : REAL
VAR_INPUT
	T : REAL;
	RH : REAL;
END_VAR
VAR CONSTANT
	CPL : REAL := 1.00482;
	CW : REAL := 1.86;
	LH : REAL := 2500.78;
END_VAR


(*
version 1.1	2 nov 2007
programmer 	hugo
tested by		tobias

this function calculates the enthalpy for humid air between 0 and 100 deg C

*)
AIR_ENTHALPY := CPL * T + (CW * T + LH) * DEW_CON(RH,T);

(* revision history

hm	31.10.2007	rev 1.0
	original version

hm	2.11.2007		rev 1.1
	deleted unused variable RF

hm	2.12.2007		rev 1.2
	changed code for better performance
*)
END_FUNCTION

(* POU Building/HLK/DEW_CON, ST *)
FUNCTION DEW_CON : REAL
VAR_INPUT
	RH : REAL;
	T : REAL;
END_VAR


(*
version 1.5	13. mar. 2009
programmer 	hugo
tested by		oscat

this function calculates the water concentratin in air for a given temperature and relative humidity.
the output states the concentration of water vapor in air in Gramms / qubic meter.

*)
(*	this code is good to read but need to be improoved
	SDD := 6.1078*EXPT(10,(a*T)/(b+T));
	DD := RH/100 * SDD;
	V := LOG(DD/6.1078);
	TD := b*V/(a-v);
	dew_con := 0.1 * mw / RU * DD / (T - TK);
*)
IF RH > 0.0 THEN
	DEW_CON := 2.166824303E-2 * RH * SDD(T,FALSE)  / (T - phys.T0);
END_IF;

(*
Bezeichnungen:
r = relative Luftfeuchte
T = Temperatur in °C
TK = Temperatur in Kelvin (TK = T + 273.15)
TD = Taupunkttemperatur in °C
DD = Dampfdruck in hPa
SDD = Sättigungsdampfdruck in hPa

Parameter:
a = 7.5, b = 237.3 für T >= 0
a = 7.6, b = 240.7 für T < 0 über Wasser (Taupunkt)
a = 9.5, b = 265.5 für T < 0 über Eis (Frostpunkt)

R* = 8314.3 J/(kmol*K) (universelle Gaskonstante)
mw = 18.016 kg (Molekulargewicht des Wasserdampfes)
AF = absolute Feuchte in g Wasserdampf pro m3 Luft

Formeln:

   1. SDD(T) = 6.1078 * 10^((a*T)/(b+T))
   2. DD(r,T) = r/100 * SDD(T)
   3. r(T,TD) = 100 * SDD(TD) / SDD(T)
   4. TD(r,T) = b*v/(a-v) mit v(r,T) = log10(DD(r,T)/6.1078)
   5. AF(r,TK) = 10^5 * mw/R* * DD(r,T)/TK; AF(TD,TK) = 10^5 * mw/R* * SDD(TD)/TK 

*)

(* revision history

hm 29 apr 2007	rev 1.0
	original version

hm	13.sep 2007	rev 1.1
	improoved coding for speed
	deleted unused variabled SDD,DD,V, TD

hm	2. dec 2007	rev 1.2
	changed code for better performance
	output is now in Gramms / Qubic meter

hm	14. oct. 2008	rev 1.3
	performance improvement

hm	18. oct. 2008	rev 1.4
	using phys constants

hm	13. mar. 2009	rev 1.5
	improved code
*)
END_FUNCTION

(* POU Engineering/measurements/ALARM_2, ST *)
FUNCTION_BLOCK ALARM_2
VAR_INPUT
	X : REAL;
	LO_1 : REAL;
	HI_1 : REAL;
	LO_2 : REAL;
	HI_2 : REAL;
	HYS : REAL;
END_VAR
VAR_OUTPUT
	Q1_LO : BOOL;
	Q1_HI : BOOL;
	Q2_LO : BOOL;
	Q2_HI : BOOL;
END_VAR
VAR
	tmp: REAL;
END_VAR

(*
	version 1.1	11. mar. 2009
	programmer 	hugo
	tested BY		tobias

ALARM_2 will check two pairs of limits and signal when the input is above or below a set limit.
with the input HYS a hysteresis can be defined for all limits. 

*)
tmp := X - Hys * 0.5;
IF tmp > LO_1 THEN Q1_LO := FALSE; END_IF;
IF tmp > LO_2 THEN Q2_LO := FALSE; END_IF;
IF tmp > HI_1 THEN Q1_HI := TRUE; END_IF;
IF tmp > HI_2 THEN Q2_HI := TRUE; END_IF;
tmp := tmp + hys;
IF tmp < LO_1 THEN Q1_LO := TRUE; END_IF;
IF tmp < LO_2 THEN Q2_LO := TRUE; END_IF;
IF tmp < HI_1 THEN Q1_HI := FALSE; END_IF;
IF tmp < HI_2 THEN Q2_HI := FALSE; END_IF;



(* revision history
hm	19. may. 2008		rev 1.0
	original version

hm	11. mar. 2009	rev 1.1
	improved code
*)
END_FUNCTION_BLOCK

(* POU Engineering/signal processing/AOUT, ST *)
FUNCTION AOUT : DWORD
VAR_INPUT
	in : REAL;
END_VAR
VAR_INPUT CONSTANT
	Bits : BYTE;
	sign : BYTE := 255;
	low : REAL;
	high : REAL := 10.0;
END_VAR
VAR CONSTANT
	ff : DWORD := 2#1;
END_VAR
VAR
	in2 : REAL;
	sx : BOOL;
END_VAR

(*
version 1.4	23 feb 2008
programmer 	oscat
tested by		tobias

this module conditions an internal real value for D/A converter.
Aout converts and internal real value to a word for an D/A converter or other output devices.
The input value is converted to a n-bit wide output and a sign bit is set separately as specified.
the outout min value is set for the specified min input value and the max output is set for the max input value.
an input higher or lower then the max or min value will set the respective max or min value or the output.


*) 
(* if sign bit is defined *)
IF sign < 32 THEN
	sx := sign_R(in);
	in2 := ABS(in);
ELSE
	in2 := in;
END_IF;

(* begrenze in auf die zulässigen werte *)
in2 := LIMIT(low, in2, high);

(* Berechne den Ausgangswert *)
Aout := REAL_TO_DWORD((in2 - low) / (high - low) * DWORD_TO_REAL(SHL(ff,bits) -1));
IF sx THEN Aout := SHL(ff,sign) OR Aout; END_IF;

(*
revision history

hm 18.1.2007		rev 1.1
	renamed Modul to aout.
	changed Output to 32 Bit max.
	corrected error with sign bit.

hm	13.9.2007		rev 1.2
	changed code to avoid warning under codesys 2.8.1

hm	2. dec 2007		rev 1.3
	changed code for better performance

hm	23. feb 2008	rev 1.4
	changed code for better performance
*)
END_FUNCTION

(* POU Mathematical/SIGN_R, ST *)
FUNCTION SIGN_R : BOOL
VAR_INPUT
	in : REAL;
END_VAR


(*
version 1.4	10. mar. 2009
programmer 	hugo
tested by		tobias

this function return true if the real input is negative

*)
SIGN_R := in < 0.0;


(* revision history
hm 19.1.2007	rev 1.1
	changed method of function for better compatibility to other systems

hm	1.12.2007	rev 1.2
	changed code to improve performance

hm	14. jun. 2008	rev 1.3
	improved performace

hm 10. mar. 2009	rev 1.4
	real constants updated to new systax using dot																																																																																																																																																																																																																																																																																																																																																																																																																																																																																																																																																																																																																																																																																																																																																																																																																																																																																																																																																																																																																																																											

*)
END_FUNCTION

(* POU Engineering/signal processing/AOUT1, ST *)
FUNCTION AOUT1 : DWORD
VAR_INPUT
	in : REAL;
END_VAR
VAR_INPUT CONSTANT
	Bit_0 : INT;
	Bit_N : INT := 31;
	sign : INT := 255;
	low : REAL;
	high : REAL := 10.0;
END_VAR
VAR CONSTANT
	ff : DWORD := 2#1;
END_VAR
VAR
	sx: BOOL;
	in2 : REAL;
END_VAR

(*
version 1.0	23 feb 2008
programmer 	oscat
tested by		tobias

this module conditions an internal real value for a D/A converter.

*) 
(* if sign bit is defined *)
IF sign < 32 THEN
	sx := SIGN_R(in);
	in2 := ABS(in);
ELSE
	in2 := in;
END_IF;

(* begrenze in auf die zulässigen werte *)
in2 := LIMIT(low, in2, high);

(* Berechne den Ausgangswert *)
AOUT1 := SHL(REAL_TO_DWORD((in2 - low) / (high - low) * DWORD_TO_REAL(SHL(ff,bit_n - Bit_0 + 1) -1)),Bit_0);
IF sx THEN AOUT1 := SHL(ff,sign) OR AOUT1; END_IF;


(* revision history
hm	23. feb 2008	rev 1.0
	original version

*)
END_FUNCTION

(* POU Mathematical/Array/ARRAY_AVG, ST *)
FUNCTION ARRAY_AVG : REAL
VAR_INPUT
	pt : POINTER TO ARRAY[0..32000] OF REAL;
	size : UINT;
END_VAR
VAR
	i: UINT;
	stop: UINT;
END_VAR

(*
version 1.3	10. mar. 2009
programmer 	hugo
tested by		tobias

this function will calculate the average of a given array.
the function needs to be called:	array_avg(adr("array"),sizeof("array"));
because this function works with pointers its very time efficient and it needs no extra memory.

*)
stop := SHR(size,2)-1;
ARRAY_AVG := pt^[0];
FOR i := 1 TO stop DO
	ARRAY_AVG := ARRAY_AVG + pt^[i];
END_FOR;
ARRAY_AVG := ARRAY_AVG / UINT_TO_REAL(stop + 1);


(* revision history
hm	2. oct 2007		rev 1.0
	original version

hm	12. dec 2007	rev 1.1
	chaged code for better performance

hm	16. mar. 2008	rev 1.2
	changed input size to uint

hm	10. mar. 2009	rev 1.3
	added type conversion for compatibility reasons
*)
END_FUNCTION

(* POU Mathematical/Array/ARRAY_GAV, ST *)
FUNCTION ARRAY_GAV : REAL
VAR_INPUT
	pt : POINTER TO ARRAY[0..32000] OF REAL;
	size : UINT;
END_VAR
VAR
	i: UINT;
	stop: UINT;
END_VAR

(*
version 1.1	10. mar. 2009
programmer 	hugo
tested by		tobias

this function will calculate the geometric average of a given array.
the function needs to be called:	array_avg(adr("array"),sizeof("array"));
because this function works with pointers its very time efficient and it needs no extra memory.

*)
stop := SHR(size,2)-1;
ARRAY_GAV := 1.0;
FOR i := 0 TO stop DO
	IF pt^[i] > 0.0 THEN
		ARRAY_GAV := ARRAY_GAV * pt^[i];
	ELSE
		ARRAY_GAV := 0.0;
		RETURN;
	END_IF;
END_FOR;
ARRAY_GAV := SQRTN(ARRAY_GAV,UINT_TO_INT(stop)+1);


(* revision history
hm	2. apr 2008	rev 1.0
	original version

hm	10. mar. 2009	rev 1.1
	real constants updated to new systax using dot

*)
END_FUNCTION

(* POU Mathematical/SQRTN, ST *)
FUNCTION SQRTN : REAL
VAR_INPUT
	X : REAL;
	N : INT;
END_VAR


(*
version 1.3	10. mar. 2009
programmer 	hugo
tested by		tobias

this function calculates the nth root function of X according to the formula sqrtn = x^(1/n).

*)
IF N > 0 THEN
	SQRTN := EXP(LN(x) / INT_TO_REAL(n));
ELSE
	SQRTN := 0.0;
END_IF;


(* revision history
hm		12 jan 2007	rev 1.0
	original version

hm		2. dec 2007	rev 1.1
	changed code for better performance

hm		11. mar 2008	rev 1.2
	added result 0 for compatibility reasons

